						CurrentSyncGroupPicking[i] :=i;
						CurrentSyncGroupPiacing[i] :=i;
					
				
						ClipsHaveNeedle_Pick[i]:=CurrentProcessdata.PickingNeedleInfo[i].CycleStart;
					//Get placing needle info	
				END_FOR
				
				FUN_GetSyncGroup_AllocationJob(Coordinates :=CurrentPickingCoordinates,NeedleInfo:=CurrentProcessData.PickingNeedleInfo, SyncGroup=>CurrentSyncGroupPicking);
				FUN_GetSyncGroup_AllocationJob(Coordinates :=CurrentPlacingCoordinates,NeedleInfo:=CurrentProcessData.PlacingNeedleInfo, SyncGroup=>CurrentSyncGroupPiacing);
				// arrange sync group in this picking/placing job
				ClipsHaveNeedle:=ClipsHaveNeedle_Pick;
				tAutoAllocationJobBatchTimeOut.IN:=FALSE;
				AllocationJobBatchMode:=E_AllocationJob.Initial;
	
			E_AllocationJob.Initial:						
				//Get All cylinders & clips back
				bCheckTrue:=TRUE;				
				tAutoAllocationJobBatchTimeOut.IN:=TRUE	;
				
				FOR i:=0 TO NrOfAllocateCylinder - 1 DO
					clips[i].M_Retract();
					IF  clips[i].InRearPosition THEN
						cylinders[i].M_Retract();		
					END_IF	
		
					IF NOT cylinders[i].InRearPosition THEN
						bCheckTrue:=FALSE;			
					END_IF
		
				END_FOR
				// recovery Axes if error occur
				bCheckTrue:=M_RecoveryAxes();
			
				IF bCheckTrue THEN	 // Only go next step if everything is fine 
					tAutoAllocationJobBatchTimeOut.IN:=FALSE	;	
					IF bAutoAllocateJobDryRun OR SimpleAllocateMode THEN //Simple allocate mode will not placing to turn table therefor no need to check boxes on turntable						
						AllocationJobBatchMode:=E_AllocationJob.CheckRotateBeltStation;
					ELSE						
						AllocationJobBatchMode:=E_AllocationJob.CheckBoxesOnTurnTableReady;
					END_IF
					
				END_IF
				IF tAutoAllocationJobBatchTimeOut.Q THEN //Timeout error
					StatusDescription :='initiial Cylindes timeout';
					uiResumableStep := E_AllocationJob.Initial;
					_Abort :=TRUE;					
				END_IF
	
	E_AllocationJob.CheckBoxesOnTurnTableReady:
		tAutoAllocationJobBatchTimeOut.IN:=TRUE	;
		bBoxCheck:=TRUE;		
				FOR i:=0 TO 3 DO
					// if R1 or R2 used in this cycle
					IF CurrentProcessdata.PlacingNeedleInfo[i].CycleStart  THEN
						IF CurrentProcessdata.PlacingNeedleInfo[i].Box=0 THEN
							R1Used :=TRUE;
							END_IF
						
						 IF  CurrentProcessdata.PlacingNeedleInfo[i].Box=1 THEN
 							R2Used :=TRUE;
						END_IF
					END_IF

				END_FOR
				
				IF  R1Used THEN 
					  bBoxCheck :=INPUT.bTurnTable_I1Detect_Sensor AND bBoxCheck; 
				END_IF
				IF  R2Used THEN 
					  bBoxCheck := INPUT.bTurnTable_I2Detect_Sensor AND bBoxCheck; 
				END_IF
 				
				IF bBoxCheck THEN
					R1Used:=FALSE;
					R2Used:=FALSE;
					bBoxCheck :=FALSE;
					IF NOT TurnTable_Press.InFrontPosition THEN
						TurnTable_Press.M_Extend();
					END_IF
					AllocationJobBatchMode:=E_AllocationJob.CheckRotateBeltStation;
				END_IF
				
				IF tAutoAllocationJobBatchTimeOut.Q THEN
					uiResumableStep := E_AllocationJob.CheckBoxesOnTurnTableReady;
					_Abort :=TRUE	;
					StatusDescription :='Box not ready on Turn table';
				END_IF
				
	E_AllocationJob.CheckRotateBeltStation:	
		// 
		tAutoAllocationJobBatchTimeOut.IN:=FALSE;
		tAutoAllocationJobBatchTimeOut.PT := T#300S;
		
		IF ClipsHaveNeedle_Pick[iWorkingIndex] THEN
				RoundBeltMoveJob.Position:=CurrentProcessData.PickingNeedleInfo[iWorkingIndex].Station;		
				// Give RoundBelt station information
				
				IF CurrentProcessData.FastMode THEN // Fast mode : XY robot will start move to picking during rotate belt moving to request station
					IF cylinders[iWorkingCylinder].InRearPosition THEN
						arAxisCtrl_gb[AxisNo.Allocate_X].PosMode.Acc := CurrentData.Axes.Allocate_X.HalfAuto.Acceleration;
						arAxisCtrl_gb[AxisNo.Allocate_X].PosMode.Dec := CurrentData.Axes.Allocate_X.HalfAuto.Deceleration;
						arAxisCtrl_gb[AxisNo.Allocate_X].PosMode.Jerk := CurrentData.Axes.Allocate_X.HalfAuto.Jerk;
						arAxisCtrl_gb[AxisNo.Allocate_X].PosMode.Velocity := CurrentData.Axes.Allocate_X.HalfAuto.Velocity;
						arAxisCtrl_gb[AxisNo.Allocate_X].PosMode.Position := CurrentPickingCoordinates[iWorkingIndex].X;
					
						arAxisCtrl_gb[AxisNo.Allocate_Y].PosMode.Acc := CurrentData.Axes.Allocate_Y.HalfAuto.Acceleration;
						arAxisCtrl_gb[AxisNo.Allocate_Y].PosMode.Dec := CurrentData.Axes.Allocate_Y.HalfAuto.Deceleration;
						arAxisCtrl_gb[AxisNo.Allocate_Y].PosMode.Jerk := CurrentData.Axes.Allocate_Y.HalfAuto.Jerk;
						arAxisCtrl_gb[AxisNo.Allocate_Y].PosMode.Velocity := CurrentData.Axes.Allocate_Y.HalfAuto.Velocity;
						arAxisCtrl_gb[AxisNo.Allocate_Y].PosMode.Position := CurrentPickingCoordinates[iWorkingIndex].Y;						
					END_IF								
				END_IF		
				AllocationJobBatchMode:=E_AllocationJob.MovingRotateBeltStation;

			ELSE				
				AllocationJobBatchMode:=E_AllocationJob.IfNextPTP_Picking;
			END_IF

            E_AllocationJob.MovingRotateBeltStation:

              RoundBeltMoveJob.HandShake.Execute := TRUE; //Internally call rotate belt to move to request station

                IF RoundBeltMoveJob.HandShake.Busy OR RoundBeltMoveJob.HandShake.Done OR bAutoAllocateJobDryRun THEN
                  AllocationJobBatchMode := E_AllocationJob.MovedRotateBeltStation;
              END_IF
			
				IF  RoundBeltMoveJob.HandShake.Error THEN
					_Error:=TRUE;
					StatusDescription := 'Allocation batch job , Rotate belt error';
				END_IF
				AllocationJobBatchMode := E_AllocationJob.MovedRotateBeltStation;
				
            E_AllocationJob.MovedRotateBeltStation:
				// wait roundbelt object
                tAutoAllocationJobBatchTimeOut.IN := TRUE;

                bMoveRotateBeltDone := RoundBeltMoveJob.HandShake.Done;
                Ton_RoundBeltArrivedDelay.IN := bMoveRotateBeltDone;

                IF bMoveRotateBeltDone OR bAutoAllocateJobDryRun THEN
                    RoundBeltMoveJob.HandShake.Execute := FALSE;
                    tAutoAllocationJobBatchTimeOut.IN := FALSE;
                    AllocationJobBatchMode := E_AllocationJob.MoveToTargetPos;
                END_IF

                IF tAutoAllocationJobBatchTimeOut.Q THEN
                    StatusDescription := 'Rotate Belt TimeOut';
                    uiResumableStep := E_AllocationJob.MovingRotateBeltStation;
                    _Abort           := TRUE;
                END_IF
				
					
            E_AllocationJob.MoveToTargetPos:
                Ton_RoundBeltArrivedDelay.IN := FALSE;
                tAutoAllocationJobBatchTimeOut.IN := TRUE;

                iWorkingCylinder :=CurrentProcessData.PickingNeedleInfo[iWorkingIndex].Clip ;

                IF NOT CurrentProcessData.FastMode THEN
					IF cylinders[iWorkingCylinder].InRearPosition THEN							
						arAxisCtrl_gb[AxisNo.Allocate_X].PosMode.Acc := CurrentData.Axes.Allocate_X.HalfAuto.Acceleration;
						arAxisCtrl_gb[AxisNo.Allocate_X].PosMode.Dec := CurrentData.Axes.Allocate_X.HalfAuto.Deceleration;
						arAxisCtrl_gb[AxisNo.Allocate_X].PosMode.Jerk := CurrentData.Axes.Allocate_X.HalfAuto.Jerk;
						arAxisCtrl_gb[AxisNo.Allocate_X].PosMode.Velocity := CurrentData.Axes.Allocate_X.HalfAuto.Velocity;
						arAxisCtrl_gb[AxisNo.Allocate_X].PosMode.Position := CurrentPickingCoordinates[iWorkingIndex].X;
					
						arAxisCtrl_gb[AxisNo.Allocate_Y].PosMode.Acc := CurrentData.Axes.Allocate_Y.HalfAuto.Acceleration;
						arAxisCtrl_gb[AxisNo.Allocate_Y].PosMode.Dec := CurrentData.Axes.Allocate_Y.HalfAuto.Deceleration;
						arAxisCtrl_gb[AxisNo.Allocate_Y].PosMode.Jerk := CurrentData.Axes.Allocate_Y.HalfAuto.Jerk;
						arAxisCtrl_gb[AxisNo.Allocate_Y].PosMode.Velocity := CurrentData.Axes.Allocate_Y.HalfAuto.Velocity;
						arAxisCtrl_gb[AxisNo.Allocate_Y].PosMode.Position := CurrentPickingCoordinates[iWorkingIndex].Y;	
					END_IF
                END_IF

                IF (arAxisCtrl_gb[AxisNo.Allocate_X].Admin.Axis.Status.Moving OR  
			(arAxisStatus_gb[AxisNo.Allocate_X].Admin._OpModeAck = ModePosAbs AND arAxisStatus_gb[AxisNo.Allocate_X].Admin.CmdDone) )AND  
					(arAxisCtrl_gb[AxisNo.Allocate_Y].Admin.Axis.Status.Moving OR 
					(arAxisStatus_gb[AxisNo.Allocate_Y].Admin._OpModeAck = ModePosAbs AND arAxisStatus_gb[AxisNo.Allocate_Y].Admin.CmdDone))
					(* AND RoundBelt.AllocatingArea.PressCylinder.InFrontPosition *) THEN
					tAutoAllocationJobBatchTimeOut.IN := FALSE;
                    AllocationJobBatchMode := E_AllocationJob.MovingToTargetPos;
                END_IF
 				
				IF arAxisCtrl_gb[AxisNo.Allocate_Y].Admin.Axis.Status.Error AND 
					arAxisCtrl_gb[AxisNo.Allocate_X].Admin.Axis.Status.Error  THEN
					_Error :=TRUE;
					StatusDescription :='Allocate robot error';
				END_IF
				
				 IF tAutoAllocationJobBatchTimeOut.Q THEN

                    StatusDescription := 'Allocate robot TimeOut';
                    uiResumableStep := E_AllocationJob.MoveToTargetPos;
                    _Abort           := TRUE;

                END_IF
				
            E_AllocationJob.MovingToTargetPos:

                tAutoAllocationJobBatchTimeOut.IN := TRUE;

                IF (arAxisStatus_gb[AxisNo.Allocate_Y].Admin._OpModeAck = ModePosAbs AND arAxisStatus_gb[AxisNo.Allocate_Y].Admin.CmdDone) AND 
					(arAxisStatus_gb[AxisNo.Allocate_X].Admin._OpModeAck = ModePosAbs AND arAxisStatus_gb[AxisNo.Allocate_X].Admin.CmdDone) THEN
                    tAutoAllocationJobBatchTimeOut.IN := FALSE;
					IF bAutoAllocateJobDryRun THEN
                   	 AllocationJobBatchMode                := E_AllocationJob.CylinderDownPick;
					ELSE
						AllocationJobBatchMode             := E_AllocationJob.CheckBoxReadyOnAllocatePosOfRoundBelt;
					END_IF
                END_IF

                IF tAutoAllocationJobBatchTimeOut.Q THEN
                    StatusDescription := 'Moving to picking position timeout';
                    uiResumableStep := E_AllocationJob.MoveToTargetPos;
                    _Abort           := TRUE;
                END_IF
				
				
			E_AllocationJob.CheckBoxReadyOnAllocatePosOfRoundBelt:
				tAutoAllocationJobBatchTimeOut.IN:=TRUE	;
				bBoxCheck :=TRUE;
				FOR i:=0 TO 3 DO //Check if request box is on the belt 
					IF CurrentProcessData.PickingNeedleInfo[i].Station =  CurrentProcessData.PickingNeedleInfo[iWorkingIndex].Station THEN
						IF CurrentProcessData.PickingNeedleInfo[i].Box=0   THEN
							A1Used :=TRUE;
							END_IF
						
						 IF  CurrentProcessData.PickingNeedleInfo[i].Box=1 THEN
 							A2Used :=TRUE;
						END_IF
					END_IF
				END_FOR
				
				IF  A1Used THEN 
					  bBoxCheck :=INPUT.bRoundBelt_WorkZoneQ1Detect_Sensor AND bBoxCheck; 
				END_IF
				IF  A2Used THEN 
					  bBoxCheck :=INPUT.bRoundBelt_WorkZoneQ2Detect_Sensor AND bBoxCheck; 
				END_IF
 				
				IF bBoxCheck THEN
						bBoxCheck:=A1Used:=A2Used:=FALSE;
						tAutoAllocationJobBatchTimeOut.IN:=FALSE	;
						IF RoundBelt_Press.InFrontPosition THEN
							AllocationJobBatchMode:=E_AllocationJob.CylinderDownPick;
						ELSE
							//RoundBelt_Press.M_Extend();	
						END_IF
				END_IF
				
				IF tAutoAllocationJobBatchTimeOut.Q THEN
					_Abort :=TRUE	;
					uiResumableStep :=E_AllocationJob.CheckBoxReadyOnAllocatePosOfRoundBelt;
					StatusDescription :='Box not ready on Rotate Belt';
				END_IF

            E_AllocationJob.CylinderDownPick:
                
                bCylinderCheck:=TRUE;
				tAutoAllocationJobBatchTimeOut.IN := TRUE;       
				
				
                THIS^.cylinders[iWorkingCylinder].M_Extend();//'AutoMode E_AllocationJob.CylinderDownPick');
				// Cylinder move down
				
				IF CurrentProcessData.SyncMode THEN
					///Sync mode : all clips in same sync group will move together to picking / placing
					FOR i := iWorkingIndex+1 TO 3 DO
						IF CurrentSyncGroupPicking[i]=CurrentSyncGroupPicking[iWorkingIndex] AND 
							ClipsHaveNeedle_Pick[i]	 THEN
							cylinders[CurrentProcessData.PickingNeedleInfo[i].Clip].M_Extend();//'Auto Mode E_AllocationJob.CylinderDownPick in Sync picking Mode');
							bCylinderCheck :=cylinders[CurrentProcessData.PickingNeedleInfo[i].Clip].InFrontPosition AND bCylinderCheck;			
						END_IF
					END_FOR
					
				END_IF
                
                IF cylinders[iWorkingCylinder].InFrontPosition AND bCylinderCheck THEN
                    tAutoAllocationJobBatchTimeOut.IN := FALSE;
                    AllocationJobBatchMode                := E_AllocationJob.ClipColse;
                END_IF

                IF tAutoAllocationJobBatchTimeOut.Q THEN

                    StatusDescription := 'Picking down timeout';
                    _Abort :=TRUE	;
					uiResumableStep :=E_AllocationJob.CylinderDownPick;

                END_IF

            E_AllocationJob.ClipColse:
                Ton_RoundBeltArrivedDelay.IN := FALSE;
                tAutoAllocationJobBatchTimeOut.IN := TRUE;
				bCylinderCheck:=TRUE;
				
                THIS^.clips[iWorkingCylinder].M_Extend();//'Auto Mode E_AllocationJob.ClipColse');
				IF CurrentProcessData.SyncMode THEN
					FOR i := iWorkingIndex+1 TO 3 DO
						IF CurrentSyncGroupPicking[i]=CurrentSyncGroupPicking[iWorkingIndex] AND 
							ClipsHaveNeedle_Pick[i]	 THEN
							clips[CurrentProcessData.PickingNeedleInfo[i].Clip].M_Extend();//'Auto Mode E_AllocationJob.ClipColse in Sync pick Mode');
							bCylinderCheck :=clips[CurrentProcessData.PickingNeedleInfo[i].Clip].InFrontPosition AND bCylinderCheck;			
						END_IF
					END_FOR
					
				END_IF
				
                IF clips[iWorkingCylinder].InFrontPosition AND bCylinderCheck THEN
                    tAutoAllocationJobBatchTimeOut.IN := FALSE;
                    AllocationJobBatchMode                := E_AllocationJob.CylinderUpPick;
                END_IF

                IF tAutoAllocationJobBatchTimeOut.Q THEN

                    StatusDescription := 'Picking Close timeout';
                    _Error := TRUE;

                END_IF

	E_AllocationJob.CylinderUpPick:
		bCylinderCheck:=TRUE;
		//bCylinderCheckFastMode:=TRUE;					
		bBoxCheck :=TRUE;
		
		tAutoAllocationJobBatchTimeOut.IN:=TRUE	;
		
		THIS^.cylinders[iWorkingCylinder].M_Retract();// 'Auto Mode E_AllocationJob.CylinderUpPick');		
		
		IF CurrentProcessData.SyncMode THEN
					FOR i := iWorkingIndex+1 TO 3 DO
						IF CurrentSyncGroupPicking[i]=CurrentSyncGroupPicking[iWorkingIndex] AND 
							ClipsHaveNeedle_Pick[i]	 THEN
							cylinders[CurrentProcessData.PickingNeedleInfo[i].Clip].M_Retract();// 'Auto Mode E_AllocationJob.CylinderUpPick in Sync pick Mode');
							bCylinderCheck :=cylinders[CurrentProcessData.PickingNeedleInfo[i].Clip].InRearPosition AND bCylinderCheck;
							//bCylinderCheckFastMode := (NOT cylinders[CurrentProcessData.PickingNeedleInfo[i].Clip].InFrontPosition) AND bCylinderCheckFastMode;
						END_IF
					END_FOR
					
		END_IF
		
				IF  A1Used THEN 
					  bBoxCheck :=INPUT.bRoundBelt_WorkZoneQ1Detect_Sensor AND bBoxCheck; 
				END_IF
				IF  A2Used THEN 
					  bBoxCheck :=INPUT.bRoundBelt_WorkZoneQ2Detect_Sensor AND bBoxCheck; 
				END_IF
				//Check if box still there
				
(*//====	2026/03/31 取消fastmode		edited by Gamin
		IF CurrentProcessData.FastMode AND bCylinderCheckFastMode AND (NOT cylinders[iWorkingCylinder].InFrontPosition) THEN
			tonFastModeTimeDelayBatch.IN:=TRUE;
		END_IF
		
		IF (cylinders[iWorkingCylinder].InRearPosition AND bCylinderCheck )OR  tonFastModeTimeDelayBatch.Q  THEN
			//Fast mode : go next step when cylinder is leave the front sensor with certain time delay
				tonFastModeTimeDelayBatch.IN:=FALSE;			
				AllocationJobBatchMode:=E_AllocationJob.IfNextPTP_Picking;
		END_IF
==========================*)
				IF cylinders[iWorkingCylinder].InRearPosition AND bCylinderCheck THEN
					AllocationJobBatchMode:=E_AllocationJob.IfNextPTP_Picking;
				END_IF

		IF tAutoAllocationJobBatchTimeOut.Q THEN			
			StatusDescription :='Picking Up timeout';
			_Abort :=TRUE	;
			uiResumableStep :=E_AllocationJob.CylinderUpPick;
		END_IF
		
	E_AllocationJob.IfNextPTP_Picking:
		tAutoAllocationJobBatchTimeOut.IN:=FALSE	;	
		iPickingNeedleCount:=1;
			FOR i := iWorkingIndex+1 TO 3 DO //remove request if already processed in previous sync group
				IF CurrentSyncGroupPicking[i]=CurrentSyncGroupPicking[iWorkingIndex] AND 
				   ClipsHaveNeedle_Pick[i]	 THEN
						iPickingNeedleCount:=iPickingNeedleCount+1;
						ClipsHaveNeedle_Pick[i]:=FALSE;		
				END_IF
			END_FOR
			
		iWorkingIndex:=iWorkingIndex+1;
		IF iWorkingIndex>= NrOfAllocateCylinder THEN //All picking job done in this cycle , go to placing processing
			iWorkingIndex:=0;
			tAutoAllocationJobBatchTimeOut.IN:=FALSE	;
			IF SimpleAllocateMode THEN //If Simple allocate mode , need to check the target box is ready on rotate belt
				AllocationJobBatchMode:=E_AllocationJob.CheckRotateBeltStation_SimpleAllocatePlacing;
			ELSE
				AllocationJobBatchMode:=E_AllocationJob.MoveToPlacingPos;
			END_IF
		ELSE
			
			AllocationJobBatchMode:=E_AllocationJob.CheckRotateBeltStation;		
			 //Still picking job
		END_IF
		
	

	E_AllocationJob.CheckRotateBeltStation_SimpleAllocatePlacing:	
		// Check if the Rotate belt is in the target.
		tAutoAllocationJobBatchTimeOut.IN:=FALSE;		
		IF ClipsHaveNeedle[iWorkingIndex] THEN
			RoundBeltMoveJob.Position:=CurrentProcessData.PlacingNeedleInfo[iWorkingIndex].Station;	
			// Give roundBelt station
			AllocationJobBatchMode:=E_AllocationJob.MovingRotateBeltStation_SimpleAllocatePlacing;
				IF CurrentProcessData.FastMode THEN // Fast mode : XY robot will start move to picking during rotate belt moving to request station
					IF cylinders[iWorkingCylinder].InRearPosition THEN				
						arAxisCtrl_gb[AxisNo.Allocate_X].PosMode.Acc := CurrentData.Axes.Allocate_X.HalfAuto.Acceleration;
						arAxisCtrl_gb[AxisNo.Allocate_X].PosMode.Dec := CurrentData.Axes.Allocate_X.HalfAuto.Deceleration;
						arAxisCtrl_gb[AxisNo.Allocate_X].PosMode.Jerk := CurrentData.Axes.Allocate_X.HalfAuto.Jerk;
						arAxisCtrl_gb[AxisNo.Allocate_X].PosMode.Velocity := CurrentData.Axes.Allocate_X.HalfAuto.Velocity;
						arAxisCtrl_gb[AxisNo.Allocate_X].PosMode.Position := CurrentPlacingCoordinates[iWorkingIndex].X;
					
						arAxisCtrl_gb[AxisNo.Allocate_Y].PosMode.Acc := CurrentData.Axes.Allocate_Y.HalfAuto.Acceleration;
						arAxisCtrl_gb[AxisNo.Allocate_Y].PosMode.Dec := CurrentData.Axes.Allocate_Y.HalfAuto.Deceleration;
						arAxisCtrl_gb[AxisNo.Allocate_Y].PosMode.Jerk := CurrentData.Axes.Allocate_Y.HalfAuto.Jerk;
						arAxisCtrl_gb[AxisNo.Allocate_Y].PosMode.Velocity := CurrentData.Axes.Allocate_Y.HalfAuto.Velocity;
						arAxisCtrl_gb[AxisNo.Allocate_Y].PosMode.Position := CurrentPlacingCoordinates[iWorkingIndex].Y;						
					END_IF							
				END_IF
		
			ELSE
				
				AllocationJobBatchMode:=E_AllocationJob.IfNextPTP_Placing;
			END_IF

            E_AllocationJob.MovingRotateBeltStation_SimpleAllocatePlacing:

                

                RoundBeltMoveJob.HandShake.Execute := TRUE; //Internally call rotate belt to move to request station

                IF RoundBeltMoveJob.HandShake.Busy OR RoundBeltMoveJob.HandShake.Done OR bAutoAllocateJobDryRun THEN
                    AllocationJobBatchMode := E_AllocationJob.MovedRotateBeltStation_SimpleAllocatePlacing;
                END_IF
				
				IF  RoundBeltMoveJob.HandShake.Error THEN
					_Error:=TRUE;
					StatusDescription := 'Allocation batch job , Rotate belt error';
				END_IF

            E_AllocationJob.MovedRotateBeltStation_SimpleAllocatePlacing:

                tAutoAllocationJobBatchTimeOut.IN := TRUE;

                bMoveRotateBeltDone := RoundBeltMoveJob.HandShake.Done;
                Ton_RoundBeltArrivedDelay.IN := bMoveRotateBeltDone;

                IF bMoveRotateBeltDone OR bAutoAllocateJobDryRun THEN
                    RoundBeltMoveJob.HandShake.Execute := FALSE;
                	tAutoAllocationJobBatchTimeOut.IN := FALSE;
                    AllocationJobBatchMode := E_AllocationJob.CheckBoxReadyOnRoundBelt_SimpleAllocateMode;
                END_IF

                IF tAutoAllocationJobBatchTimeOut.Q THEN
                    StatusDescription := 'Rotate Belt TimeOut';
                    uiResumableStep := E_AllocationJob.MovingRotateBeltStation_SimpleAllocatePlacing;
                    _Abort           := TRUE;
                END_IF
				
	E_AllocationJob.CheckBoxReadyOnRoundBelt_SimpleAllocateMode:
		tAutoAllocationJobBatchTimeOut.IN:=TRUE	;
				bBoxCheck :=TRUE;
				FOR i:=0 TO 3 DO //Check if request box is on the belt 					
						IF CurrentProcessData.PlacingNeedleInfo[i].Box=0   THEN
							A1Used :=TRUE;
							END_IF
						
						 IF  CurrentProcessData.PlacingNeedleInfo[i].Box=1 THEN
 							A2Used :=TRUE;
						END_IF
					
				END_FOR
				
				IF  A1Used THEN 
					  bBoxCheck :=INPUT.bRoundBelt_WorkZoneQ1Detect_Sensor AND bBoxCheck; 
				END_IF
				IF  A2Used THEN 
					  bBoxCheck :=INPUT.bRoundBelt_WorkZoneQ2Detect_Sensor AND bBoxCheck; 
				END_IF
 				
				IF bBoxCheck THEN
						bBoxCheck:=A1Used:=A2Used:=FALSE;
						tAutoAllocationJobBatchTimeOut.IN:=FALSE;
						AllocationJobBatchMode:=E_AllocationJob.MoveToPlacingPos;
				END_IF
				
				IF tAutoAllocationJobBatchTimeOut.Q THEN
					_Abort :=TRUE	;
					uiResumableStep :=E_AllocationJob.CheckBoxReadyOnRoundBelt_SimpleAllocateMode;
					StatusDescription :='Box not ready on Rotate Belt ';
				END_IF			
	
     E_AllocationJob.MoveToPlacingPos:
                
				tAutoAllocationJobBatchTimeOut.IN:=TRUE;
                IF ClipsHaveNeedle[iWorkingIndex] THEN 
                    iWorkingCylinder := CurrentProcessData.PlacingNeedleInfo[iWorkingIndex].Clip;
					IF cylinders[iWorkingCylinder].InRearPosition THEN
						arAxisCtrl_gb[AxisNo.Allocate_X].PosMode.Acc := CurrentData.Axes.Allocate_X.HalfAuto.Acceleration;
						arAxisCtrl_gb[AxisNo.Allocate_X].PosMode.Dec := CurrentData.Axes.Allocate_X.HalfAuto.Deceleration;
						arAxisCtrl_gb[AxisNo.Allocate_X].PosMode.Jerk := CurrentData.Axes.Allocate_X.HalfAuto.Jerk;
						arAxisCtrl_gb[AxisNo.Allocate_X].PosMode.Velocity := CurrentData.Axes.Allocate_X.HalfAuto.Velocity;
						arAxisCtrl_gb[AxisNo.Allocate_X].PosMode.Position := CurrentPlacingCoordinates[iWorkingIndex].X;
					
						arAxisCtrl_gb[AxisNo.Allocate_Y].PosMode.Acc := CurrentData.Axes.Allocate_Y.HalfAuto.Acceleration;
						arAxisCtrl_gb[AxisNo.Allocate_Y].PosMode.Dec := CurrentData.Axes.Allocate_Y.HalfAuto.Deceleration;
						arAxisCtrl_gb[AxisNo.Allocate_Y].PosMode.Jerk := CurrentData.Axes.Allocate_Y.HalfAuto.Jerk;
						arAxisCtrl_gb[AxisNo.Allocate_Y].PosMode.Velocity := CurrentData.Axes.Allocate_Y.HalfAuto.Velocity;
						arAxisCtrl_gb[AxisNo.Allocate_Y].PosMode.Position := CurrentPlacingCoordinates[iWorkingIndex].Y;						
					END_IF
							
					IF CurrentProcessData.FastMode AND NOT SimpleAllocateMode THEN // Fast mode : When robot go to placing needles , Rotatebelt will start to move to next picking station	But not allow in simple allocate job due to placing location is rotatebelt also					
						IF AutoAllocateJobBatch_Ctrl.AutoMode_AllocateMoveBatch.NrOfAllocationJob > iProcessingIndex+1 THEN//AND AutoAllocateJobBatch_Ctrl.AutoMode_AllocateMoveBatch.AllocationInfo[iProcessingIndex+1]. <> iCurrentRotateBeltStation THEN
							FOR i := 0 TO 3 DO 
								IF	AutoAllocateJobBatch_Ctrl.AutoMode_AllocateMoveBatch.AllocationInfo[iProcessingIndex+1].PickingNeedleInfo[i].CycleStart THEN
									iNextPickingStation :=   AutoAllocateJobBatch_Ctrl.AutoMode_AllocateMoveBatch.AllocationInfo[iProcessingIndex+1].PickingNeedleInfo[i].Station;
									bIfNextCycle:=TRUE;
									EXIT;
								END_IF
							END_FOR
						END_IF					
					END_IF							
							

                    IF (arAxisCtrl_gb[AxisNo.Allocate_X].Admin.Axis.Status.Moving AND  arAxisCtrl_gb[AxisNo.Allocate_Y].Admin.Axis.Status.Moving) OR
 						(arAxisStatus_gb[AxisNo.Allocate_X].Admin._OpModeAck = ModePosAbs AND arAxisStatus_gb[AxisNo.Allocate_X].Admin.CmdDone) AND 
						(arAxisStatus_gb[AxisNo.Allocate_Y].Admin._OpModeAck = ModePosAbs AND arAxisStatus_gb[AxisNo.Allocate_Y].Admin.CmdDone) THEN
						bIfNextCycle :=FALSE;
						tAutoAllocationJobBatchTimeOut.IN:=FALSE	;
                        AllocationJobBatchMode := E_AllocationJob.MovingToPlacingPos;
                    END_IF

                ELSE

                    AllocationJobBatchMode := E_AllocationJob.IfNextPTP_Placing;
                END_IF
				
				IF tAutoAllocationJobBatchTimeOut.Q THEN
			
					StatusDescription :='Move to placing timeout';
					uiResumableStep := E_AllocationJob.MoveToPlacingPos;
					_Abort := TRUE;
					
				END_IF

            E_AllocationJob.MovingToPlacingPos:

                tAutoAllocationJobBatchTimeOut.IN := TRUE;

					IF (arAxisStatus_gb[AxisNo.Allocate_X].Admin._OpModeAck = ModePosAbs AND arAxisStatus_gb[AxisNo.Allocate_X].Admin.CmdDone) AND 
						(arAxisStatus_gb[AxisNo.Allocate_Y].Admin._OpModeAck = ModePosAbs AND arAxisStatus_gb[AxisNo.Allocate_Y].Admin.CmdDone) THEN
                    tAutoAllocationJobBatchTimeOut.PT := T#300S;
                    tAutoAllocationJobBatchTimeOut.IN := FALSE;
                    AllocationJobBatchMode                := E_AllocationJob.CylinderDownPlace;
                END_IF

                IF tAutoAllocationJobBatchTimeOut.Q THEN
                    StatusDescription := 'Moving placing timeout';
                    uiResumableStep := E_AllocationJob.MoveToPlacingPos;
                    _Abort           := TRUE;

                END_IF

            E_AllocationJob.CylinderDownPlace:
				bCylinderCheck:=TRUE;
                tAutoAllocationJobBatchTimeOut.IN := TRUE;
                cylinders[iWorkingCylinder].M_Extend();//'Auto Mode E_AllocationJob.CylinderDownPlace');
				
				IF CurrentProcessData.SyncMode THEN
					FOR i := iWorkingIndex+1 TO 3 DO
						IF CurrentSyncGroupPiacing[i]=CurrentSyncGroupPiacing[iWorkingIndex] AND 
							ClipsHaveNeedle[i]	 THEN
							cylinders[CurrentProcessData.PlacingNeedleInfo[i].Clip].M_Extend();//'Auto Mode E_AllocationJob.CylinderDownPlace in Sync placing Mode');
							bCylinderCheck :=cylinders[CurrentProcessData.PlacingNeedleInfo[i].Clip ].InFrontPosition AND bCylinderCheck;			
						END_IF
					END_FOR
					
				END_IF
				
               	 IF cylinders[iWorkingCylinder].InFrontPosition AND bCylinderCheck THEN
                    tAutoAllocationJobBatchTimeOut.IN := FALSE;
                    AllocationJobBatchMode            := E_AllocationJob.ClipOpen;
              	  END_IF
				
                IF tAutoAllocationJobBatchTimeOut.Q THEN

                    StatusDescription := ' placing down timeout';
                   _Abort :=TRUE	;
					uiResumableStep :=E_AllocationJob.CylinderDownPlace;

                END_IF

            E_AllocationJob.ClipOpen:
                tAutoAllocationJobBatchTimeOut.IN := TRUE;
				bCylinderCheck:=TRUE;
                clips[iWorkingCylinder].M_Retract();// 'Auto Mode E_AllocationJob.ClipOpen');
					IF CurrentProcessData.SyncMode THEN
					FOR i := iWorkingIndex+1 TO 3 DO
						IF CurrentSyncGroupPiacing[i]=CurrentSyncGroupPiacing[iWorkingIndex] AND 
							ClipsHaveNeedle[i]	 THEN
							clips[CurrentProcessData.PlacingNeedleInfo[i].Clip].M_Retract();// 'Auto Mode E_AllocationJob.ClipOpen in Sync placing Mode');
							bCylinderCheck :=clips[CurrentProcessData.PlacingNeedleInfo[i].Clip].InRearPosition AND bCylinderCheck;			
						END_IF
					END_FOR
					
				END_IF
				
				
                IF clips[iWorkingCylinder].InRearPosition AND bCylinderCheck THEN
                    tAutoAllocationJobBatchTimeOut.IN := FALSE;
                    AllocationJobBatchMode                := E_AllocationJob.CylinderUpPlace;
                END_IF

                IF tAutoAllocationJobBatchTimeOut.Q THEN

                    StatusDescription := ' placing Open timeout';
                    _Error := TRUE;

                END_IF

            E_AllocationJob.CylinderUpPlace:
				bCylinderCheck:=TRUE;
				//bCylinderCheckFastMode:=TRUE;
				tAutoAllocationJobBatchTimeOut.IN:=TRUE;
				
                cylinders[iWorkingCylinder].M_Retract();// ' Auto Mode E_AllocationJob.CylinderUpPlace');
				
					IF CurrentProcessData.SyncMode THEN
					FOR i := iWorkingIndex+1 TO 3 DO
						IF CurrentSyncGroupPiacing[i]=CurrentSyncGroupPiacing[iWorkingIndex] AND 
							ClipsHaveNeedle[i]	 THEN
							cylinders[CurrentProcessData.PlacingNeedleInfo[i].Clip].M_Retract();// 'Auto Mode E_AllocationJob.CylinderUpPlace in Sync placing Mode');
							bCylinderCheck :=cylinders[CurrentProcessData.PlacingNeedleInfo[i].Clip ].InRearPosition AND bCylinderCheck;	
							//bCylinderCheckFastMode := (NOT cylinders[CurrentProcessData.PlacingNeedleInfo[i].Clip ].InFrontPosition) AND bCylinderCheckFastMode ;
							
						END_IF
					END_FOR					
				END_IF
(*================	取消 fastmode，防止偷跑導致撞機，edited BY Gamin 2026/03/31
				IF CurrentProcessData.FastMode  AND (NOT cylinders[iWorkingCylinder].InFrontPosition) AND bCylinderCheckFastMode THEN						
               		 tonFastModeTimeDelayBatch.IN := TRUE;
				END_IF
				
                IF (cylinders[iWorkingCylinder].InRearPosition AND bCylinderCheck) OR tonFastModeTimeDelayBatch.Q THEN
                    tAutoAllocationJobBatchTimeOut.IN         := FALSE;
					tonFastModeTimeDelayBatch.IN 				  := FALSE;
                    
                    AllocationJobBatchMode := E_AllocationJob.CheckNeedlePlaced;
                END_IF
====================*)
				IF cylinders[iWorkingCylinder].InRearPosition AND bCylinderCheck THEN
                    tAutoAllocationJobBatchTimeOut.IN         := FALSE;
                    AllocationJobBatchMode := E_AllocationJob.CheckNeedlePlaced;
                END_IF
				
                IF tAutoAllocationJobBatchTimeOut.Q THEN

                    StatusDescription := ' placing Up timeout';
                    _Abort :=TRUE	;
					uiResumableStep :=E_AllocationJob.CylinderUpPlace;

                END_IF

			E_AllocationJob.CheckNeedlePlaced:
				ClipsHaveNeedle[iWorkingIndex] :=FALSE;
					IF CurrentProcessData.SyncMode THEN
					FOR i := iWorkingIndex+1 TO 3 DO
						IF CurrentSyncGroupPiacing[i]=CurrentSyncGroupPiacing[iWorkingIndex] AND 
							ClipsHaveNeedle[i]	 THEN
							ClipsHaveNeedle[i]:=FALSE;
							
						END_IF
					END_FOR		
				END_IF
				
				
				AllocationJobBatchMode := E_AllocationJob.IfNextPTP_Placing;
				
            E_AllocationJob.IfNextPTP_Placing:
                iWorkingIndex := iWorkingIndex + 1;

                IF iWorkingIndex >= NrOfAllocateCylinder THEN
                    iWorkingIndex := 0;
                    AllocationJobBatchMode := E_AllocationJob.Finish;
                ELSE
					IF SimpleAllocateMode THEN
						AllocationJobBatchMode := E_AllocationJob.CheckRotateBeltStation_SimpleAllocatePlacing;
					ELSE
                    	AllocationJobBatchMode := E_AllocationJob.MoveToPlacingPos;
               	 END_IF
				END_IF        

            E_AllocationJob.Finish:
                // Finish
					//Update needling data
					arrProcessedIndex[iProcessingIndex] :=CurrentProcessData.ID;
				IF 	AutoAllocateJobBatch_Ctrl.AutoMode_AllocateMoveBatch.NrOfAllocationJob> iProcessingIndex THEN

					iProcessingIndex :=iProcessingIndex+1;
					AllocationJobBatchMode := E_AllocationJob.PreDataProcess;
				ELSE
					// 最後一筆邏輯完成,但機械可能還在收尾。
					// 進入 FinalCleanup gate,等所有 cylinder/clip/press 都歸位、RoundBelt idle 才設 _Executed
					AllocationJobBatchMode := E_AllocationJob.FinalCleanup;
				END_IF

			E_AllocationJob.FinalCleanup:
				// 給 Done 之前的最終收尾 gate:
				// 確保整批做完後,所有 cylinder/clip 都退到安全位置、RoundBelt 不再 Busy,
				// 才允許 _Executed := TRUE → STATE_DONE。
				// 目的: 上位看到 Done 時、PLC 內部資料(ProcessedIndex/WorkedID)跟機械都已穩定,
				//       上位撤 Execute 後即使馬上下一包進來也不會撞到上一包未收尾的狀態。
				// 註: TurnTable_Press / RoundBelt_Press 不收 — 兩個 Press 只是壓住盒子,
				//     對下一批的 X/Y robot 跟 cylinder 升降都沒有安全顧慮;
				//     收了反而會讓盒子晃動,且下一批 CheckBoxesOnTurnTableReady 還要再 Extend。
				tAutoAllocationJobBatchTimeOut(IN := TRUE, PT := T#10S);
				bCheckTrue := TRUE;

				FOR i := 0 TO NrOfAllocateCylinder-1 DO
					clips[i].M_Retract();
					IF clips[i].InRearPosition THEN
						cylinders[i].M_Retract();
					END_IF
					IF NOT cylinders[i].InRearPosition OR NOT clips[i].InRearPosition THEN
						bCheckTrue := FALSE;
					END_IF
				END_FOR

				// 圓帶不可還在動作中
				IF RoundBeltMoveJob_Status.Busy THEN
					bCheckTrue := FALSE;
				END_IF

				// 同步把最後一筆 ID 確實出到 ProcessedIndex (頂部已每 cycle 拷貝,這裡是雙保險)
				ProcessedIndex := arrProcessedIndex;

				IF bCheckTrue THEN
					tAutoAllocationJobBatchTimeOut.IN := FALSE;
					_Executed := TRUE;
				END_IF

				IF tAutoAllocationJobBatchTimeOut.Q THEN
					StatusDescription := 'FinalCleanup timeout: hardware not back to safe position';
					_UniqueErrorCode := 'E_FINAL_CLEANUP_TIMEOUT';
					uiResumableStep := E_AllocationJob.FinalCleanup;
					_Abort := TRUE;
				END_IF

        END_CASE

IF NOT Execute THEN
	eState:=STATE_RESETTING;
END_IF
IF _Error THEN
	eState:=STATE_ERROR;
END_IF
IF _Abort THEN
	eSTATE:=STATE_ABORTING;
END_IF
IF _Executed THEN
	eSTATE:=STATE_Done;
END_IF
END_METHOD

METHOD  M_STATE_RESETTING
VAR_INPUT
END_VAR
VAR	
	bCylinderCheck : BOOL;
END_VAR
Busy                         := TRUE;
Error                        := _Error;
tAutoAllocationJobBatchTimeOut.IN := FALSE;

  CASE uiResettingStep OF
            0:
                // Resetting process start

                uiAbortingStep := 0;
                uiAbortedStep  := 0;
				_bRetry := FALSE;
				RoundBeltMoveJob.HandShake.Execute:=FALSE;
				RoundBeltMoveJob_Ctrl.Execute:= RoundBeltMoveJob.HandShake.Execute;
				DAS_CoreSys.MachineControl.fbAllocateArea.M_ReleaseRoundBeltAccess(E_RoundBeltControlAccess.Allocating);

                IF M_RecoveryAxes() THEN
					uiResettingStep := 1000;
				END_IF

            1000:
				bCylinderCheck :=TRUE;
//                FOR i := 1 TO 3 DO
//                    IF cylinders[i].xError THEN
//                         cylinders[i].M_Reset();
//						 ELSE
//						 cylinders[i].M_Retract();
//                    END_IF
//				bCylinderCheck := bCylinderCheck AND cylinders[i].InRearPosition;

//                END_FOR
				RoundBeltMoveJob.HandShake.Execute:=FALSE;
				RoundBeltMoveJob_Ctrl.Execute:= RoundBeltMoveJob.HandShake.Execute;
				DAS_CoreSys.MachineControl.fbAllocateArea.M_ReleaseRoundBeltAccess(E_RoundBeltControlAccess.Allocating);
                uiResettingStep := 2000;

			2000:
//					IF TurnTable.Motor.Error THEN
//					TurnTable.Motor.Reset();
//				END_IF

//				IF  AllocateRobot.axX.Error THEN
//					  AllocateRobot.axX.Reset();
//				END_IF

//				IF  AllocateRobot.axY.Error THEN
//					  AllocateRobot.axY.Reset();
//				END_IF

//				IF RoundBelt.Motor.Error THEN
//					RoundBelt.Motor.Reset();
//				END_IF
				uiResettingStep := 9000;

            9000:
                // Resetting process is finished
                Done := FALSE;
                Busy := FALSE;
                bResettingCompleted := TRUE;
        END_CASE

        IF bResettingCompleted THEN
            eState := STATE_DORMANT;
        END_IF
END_METHOD

END_FUNCTION_BLOCK

// ---- POUs/DAS_CoreSys.TcPOU
PROGRAM DAS_CoreSys
VAR
    UserModeCofig  : PML_UnitModeConfig; //User can configure his own Mode
    MachineControl : FB_MachineControl;
	CoreSys_Stop : BOOL;
	CoreSys_Reset :BOOL;
	CoreSys_Start : BOOL;
	CoreSys_Estop : BOOL;
	OP_Mode : E_UnitMode := E_UnitMode.Manual;
	trigResetForRS485 : R_TRIG;
END_VAR

A00_BasicUnit();
A10_StatusCtrl();


CASE GVL_ADS.MachineMode.TargetMode OF
		E_MachineMode.MANUAL:
			OP_Mode := E_UnitMode.Manual;
		E_MachineMode.AUTO:
			OP_Mode := E_UnitMode.Auto;
ELSE
	OP_Mode := E_UnitMode.Manual;
END_CASE


//IF OP_Mode = E_UnitMode.Manual THEN
//	GVL_ADS.MachineMode.CurrentMode := E_MachineMode.MANUAL;
//ELSIF OP_Mode = E_UnitMode.Auto AND MachineControl.MachineHomed THEN
	
//	GVL_ADS.MachineMode.CurrentMode := E_MachineMode.AUTO;
//END_IF

IF PackTags[0].Status.UnitModeCurrent = E_UnitMode.Manual THEN
	GVL_ADS.MachineMode.CurrentMode := E_MachineMode.MANUAL;
ELSIF PackTags[0].Status.UnitModeCurrent = E_UnitMode.Auto THEN
	GVL_ADS.MachineMode.CurrentMode := E_MachineMode.AUTO;
END_IF

ACTION A00_BasicUnit:
CoreSys_Start := MachineControl.Machine_Start;
CoreSys_Stop := MachineControl.Machine_Stop;
CoreSys_Reset := MachineControl.Machine_Reset;
MachineControl(
    eModeCommand := PackTags[0].Command.UnitMode,
    eStateCommand := PackTags[0].Command.CntrlCmd,
    PackTag := PackTags[0],
    INPUT := GVL_Input.uniDI.stDI,
    OUTPUT := GVL_Output.uniDO.stDO); // FB_MachineControl
PackTags[0].Status.StateCurrent := MachineControl.eStateCurrent;
PackTags[0].Status.UnitModeCurrent := MachineControl.eModeCurrent;
CoreSys_Estop := MachineControl.Machine_Estop;
END_ACTION

ACTION A01_UnitModeConfig:
//UserModeCofig(
//	eMode							:= ePMLUnitMode_Service, 
//	bDisableClearing				:= TRUE, 
//	bDisableStarting				:= TRUE, 
//	bDisableSuspended				:= FALSE, 
//	bDisableStopping				:= TRUE, 
//	bDisableAborting				:= TRUE, 
//	bDisableHolding					:= TRUE, 
//	bDisableHeld					:= TRUE, 
//	bDisableUnholding				:= TRUE, 
//	bDisableSuspending				:= TRUE, 
//	bDisableUnsuspending			:= TRUE, 
//	bDisableResetting				:= TRUE, 
//	bDisableIdle					:= TRUE, 
//	bDisableCompleting				:= TRUE, 
//	bDisableComplete				:= TRUE, 
//	bEnableUnitModeChangeStopped	:= TRUE, 
//	bEnableUnitModeChangeIdle		:= FALSE, 
//	bEnableUnitModeChangeSuspended	:= FALSE, 
//	bEnableUnitModeChangeExecute	:= FALSE, 
//	bEnableUnitModeChangeAborted	:= TRUE, 
//	bEnableUnitModeChangeHeld		:= FALSE, 
//	bEnableUnitModeChangeComplete	:= FALSE, 
//	bError							=> , 
//	nErrorId						=> );
END_ACTION

ACTION A10_StatusCtrl:
IF PackTags[0].Status.UnitModeCurrent = E_UnitMode.Manual THEN
	IF PackTags[0].Status.StateCurrent = ePMLState_Aborted AND NOT MachineControl.Error THEN
		PackTags[0].Command.CntrlCmd := ePMLCommand_Clear;
	END_IF
	IF PackTags[0].Status.StateCurrent = ePMLState_Stopped THEN
		IF OP_Mode = E_UnitMode.Manual THEN
		PackTags[0].Command.CntrlCmd := ePMLCommand_Reset;
		END_IF
	END_IF
	IF PackTags[0].Status.StateCurrent = ePMLState_Idle THEN
		PackTags[0].Command.CntrlCmd := ePMLCommand_Start;
	END_IF
ELSIF PackTags[0].Status.UnitModeCurrent = E_UnitMode.Auto THEN
	IF PackTags[0].Status.StateCurrent = ePMLState_Aborted AND NOT MachineControl.Error THEN
		PackTags[0].Command.CntrlCmd := ePMLCommand_Clear;
	END_IF
	IF PackTags[0].Status.StateCurrent = ePMLState_Stopped THEN
		IF OP_Mode = E_UnitMode.Auto THEN
		PackTags[0].Command.CntrlCmd := ePMLCommand_Reset;
		END_IF
	END_IF
	IF PackTags[0].Status.StateCurrent = ePMLState_Idle THEN
		PackTags[0].Command.CntrlCmd := ePMLCommand_Start;
	END_IF
END_IF

IF PackTags[0].Status.UnitModeCurrent = E_UnitMode.Manual THEN
    IF ((PackTags[0].Status.StateCurrent = ePMLState_Stopped) OR
        (PackTags[0].Status.StateCurrent = ePMLState_Aborted) OR
        (PackTags[0].Status.StateCurrent = ePMLState_Execute)) AND
        MachineControl.MachineHomed
        THEN
        IF OP_Mode = E_UnitMode.Auto THEN
            PackTags[0].Command.UnitMode := E_UnitMode.Auto;
			IF PackTags[0].Status.StateCurrent = ePMLState_Execute THEN
				PackTags[0].Command.CntrlCmd := ePMLCommand_Stop;
			END_IF
        END_IF
    END_IF
ELSIF PackTags[0].Status.UnitModeCurrent = E_UnitMode.Auto THEN
    IF ((PackTags[0].Status.StateCurrent = ePMLState_Stopped) OR
        (PackTags[0].Status.StateCurrent = ePMLState_Aborted) OR
        (PackTags[0].Status.StateCurrent = ePMLState_Execute))
        THEN
        IF OP_Mode = E_UnitMode.Manual THEN
			IF PackTags[0].Status.StateCurrent <> ePMLState_Aborted OR PackTags[0].Status.StateCurrent <> ePMLState_Aborting THEN
				PackTags[0].Command.CntrlCmd := ePMLCommand_Abort;
			END_IF
            PackTags[0].Command.UnitMode := E_UnitMode.Manual;
        END_IF
    END_IF
END_IF

//GVL_ADS.OpPannel_Status.EStopBtnStatus := CoreSys_Estop;
//GVL_ADS.OpPannel_Status.ResetBtnStatus := CoreSys_Reset;
//GVL_ADS.OpPannel_Status.StartBtnStatus := CoreSys_Start;
//GVL_ADS.OpPannel_Status.StopBtnStatus := CoreSys_Stop;
// Start
IF PackTags[0].Status.UnitModeCurrent = E_UnitMode.Auto THEN
	CASE PackTags[0].Status.StateCurrent OF
		ePMLState_Idle:
			IF CoreSys_Start THEN
				PackTags[0].Command.CntrlCmd := ePMLCommand_Start;
			END_IF
	END_CASE
END_IF

// Reset & Clear

IF PackTags[0].Status.UnitModeCurrent = E_UnitMode.Auto THEN
	CASE PackTags[0].Status.StateCurrent OF
		ePMLState_Stopped,ePMLState_Complete:
			IF CoreSys_Reset THEN
				PackTags[0].Command.CntrlCmd := ePMLCommand_Reset;
			END_IF
		ePMLState_Aborted:
			IF CoreSys_Reset THEN
				PackTags[0].Command.CntrlCmd := ePMLCommand_Clear;
			END_IF
		ePMLState_Held:
			IF CoreSys_Reset THEN
				PackTags[0].Command.CntrlCmd := ePMLCommand_Unhold;
			END_IF
		ePMLState_Suspended:
			IF CoreSys_Reset THEN
				PackTags[0].Command.CntrlCmd := ePMLCommand_Unsuspend;
			END_IF
	END_CASE
END_IF

// === 光電板斷點重啟 ===
// 按 Reset 時若有 851~854 alarm,順便 power cycle Y10.5/Y10.6,
// 合併到既有 Reset 流程,不用操作員另外去找 Reboot Modbus 按鈕。
// R_TRIG 抓上升緣 + Status.Busy 雙重保險避免連續觸發。
trigResetForRS485(CLK := CoreSys_Reset);
IF trigResetForRS485.Q AND
   (   (MAIN2_RS485.RS485_V2[1].bError AND NOT GVL_HMI.Setup.Mechanical.stModbusByPass.switchOff_1)
    OR (MAIN2_RS485.RS485_V2[2].bError AND NOT GVL_HMI.Setup.Mechanical.stModbusByPass.switchOff_2)
    OR (MAIN2_RS485.RS485_V2[3].bError AND NOT GVL_HMI.Setup.Mechanical.stModbusByPass.switchOff_3)
    OR (MAIN2_RS485.RS485_V2[4].bError AND NOT GVL_HMI.Setup.Mechanical.stModbusByPass.switchOff_4))
   AND NOT GVL_ADS.RebootModbusDevices.Status.Busy
THEN
    GVL_ADS.RebootModbusDevices.Command.Execute := TRUE;
END_IF

// reboot 完成自動清 Execute,讓下次 Reset 還能觸發
IF GVL_ADS.RebootModbusDevices.Status.Done THEN
    GVL_ADS.RebootModbusDevices.Command.Execute := FALSE;
END_IF

 //Stop

IF PackTags[0].Status.UnitModeCurrent = E_UnitMode.Auto THEN
	CASE PackTags[0].Status.StateCurrent OF
		ePMLState_Execute:
			IF CoreSys_Stop THEN
				PackTags[0].Command.CntrlCmd := ePMLCommand_Suspend;
			END_IF
	END_CASE
END_IF
END_ACTION

END_PROGRAM

// ---- Library/20_MachineUnits/22_AllocateArea/Service/FB_AllocateMoveAutoBatchMode_Reverse.TcPOU
FUNCTION_BLOCK FB_AllocateMoveAutoBatchMode_Reverse EXTENDS FB_ObjectBase_V2
VAR_INPUT
//    Execute    :BOOL;   // True : This prog will start.
//    Abort      :BOOL;   // True : This prog will be abort.
//    Reset      :BOOL;   // True : This prog will be reset.
//    ObjectName :STRING; // Set this fb name(About it's action)
//	  Pause		 :BOOL;
	bOccupied							: BOOL;	
	Clips 								: REFERENCE TO  ARRAY[0..3] OF FB_Cylinder;
	cylinders 							: REFERENCE TO  ARRAY[0..3] OF FB_Cylinder;	
	TurnTable_Press		 		   		: REFERENCE TO FB_Cylinder;
	RoundBelt_Press 			   		: REFERENCE TO FB_Cylinder;
	AutoAllocateJobBatch_Reverse_Ctrl   :st_AllocateMoveAutoBatchMode_Ctrl;
	INPUT            			   		: REFERENCE TO ST_InputTable;
    OUTPUT           			   		: REFERENCE TO ST_OutputTable;
	NrOfAllocateCylinder 		   		: INT :=4;
	CurrentData 				   		: REFERENCE TO ST_SetupPara; // Componets setup parameter
	bAutoAllocateJobDryRun         		: BOOL := FALSE;
	RoundBeltMoveJob_Status 			: ST_StatusBasic;
END_VAR

VAR_OUTPUT
//    Busy    :BOOL;        // True : This prog is running.
//    Done    :BOOL;        // True : Command has been executed.
//    Aborted :BOOL;        // True : This prog is aborted.
//    Error   :BOOL;        // True : This prog has an error.
//    ErrorID :UINT;       // Output ErrorID
//    Status  :T_MaxString; // Output this prog status by string(255bytes)
	RoundBeltMoveJob_Ctrl : ST_CommandBasic;
	ProcessedIndex : ARRAY[0..49] OF INT;
	//UniqueErrorCode :STRING;
	// AutoAllocateJobBatch_Status    :st_AllocateMoveAutoBatchMode_Status;
	RoundBeltMoveJob_Position	:LREAL;
	bAllocateRobotMoveRequest : BOOL;
END_VAR

VAR
//    eState :E_MethodStatus_Basic;
//	uiExecutingStep : UDINT; // This var is used to been controll STATE_EXECUTING process.
//	uiResettingStep : UDINT;
//	uiAbortingStep : UDINT;
//	_Executed :BOOL; // Executing process completed.
//	_Error : BOOL; // FB has an error.
//	_ResetCompleted : BOOL; // FB resetting completed.
//	_AbortCompleted : BOOL; // FB aborting completed.
//	_Abort		: BOOL;
	strStatus	: STRING;
	uiResumeStep : UINT;

//	bSimpleAllocationBatchEnable		 :BOOL;
//	AutoRotatebelt_Internal_Ctrl   : st_RoundBeltAutoSingleMove_Ctrl;
	_UniqueErrorCode : STRING;
	arrProcessedIndex : ARRAY[0..49] OF INT;
 //   eState              :E_MethodStatus_Basic;  
  //  uiAbortingStep      :UDINT;
    uiAbortedStep       :UDINT;
  //  uiResettingStep     :UDINT;
	uiResumableStep		: E_AllocationJob;
    bAborttingCompleted :BOOL; // True: Aborting process finished
    bAborted            :BOOL; // True : Aborted process finished
    bExecuted           :BOOL; // True : Executing process finished
    bResettingCompleted :BOOL; // True : Resetting process finished  
    iWorkingIndex		:UINT:=0;	
	iProcessingIndex	:INT :=0;
	iWorkingCylinder	:INT;
	//_Error				:BOOL :=FALSE;
	StatusDescription	:STRING;
	ClipsHaveNeedle		: ARRAY[0..3] OF BOOL;
	ClipsHaveNeedle_Pick		: ARRAY[0..3] OF BOOL;
	ClipsHaveNoNeedle	: ARRAY[0..3] OF BOOL;
	bCylinderCheck 		: BOOL;
	bCylinderCheckFastMode : BOOL;
	iPickingNeedleCount		:INT;
	iPlacingNeedleCount		:INT;
	bIfNextCycle			:BOOL;
	bCheckStation			:BOOL:=FALSE;
	
	
	
	tAutoAllocationJobBatchTimeOut_Reverse:Tc2_Standard.TON;
    sAllocationJobBatchStatus      :STRING;
    tonFastModeTimeDelayBatch_Reverse      :Tc2_Standard.TON;
	AllocationJobBatchModeReverse		:E_AllocationJob := E_AllocationJob.Defult;
	 Ton_RoundBeltArrivedDelay     : TON;
	 CurrentPosition : ST_PositionTable;
	
  	RoundBeltMoveJob : st_AllocateCircleMoveStructure;	
		
//==========================M_AllocationJobBatchMode================================

	{attribute 'hide'}
	bCheckTrue : BOOL:=TRUE;
	iCurrentRotateBeltStation : UINT;
	i : UINT;	
	j : UINT;	

	bMoveRotateBeltBusy	:BOOL;
	bMoveRotateBeltDone : BOOL;
	A1Used				:BOOL :=FALSE;
	A2Used				:BOOL :=FALSE;
	R1Used				:BOOL :=FALSE;
	R2Used				:BOOL :=FALSE;
	bBoxCheck			:BOOL :=TRUE;
	PickingStation		:UINT;
	iNextPickingStation :UINT;
	
	_bRetry : BOOL;

	
	
END_VAR

A00_BasicUnits();
SUPER^.A10_StateControl();

(*============================================================
Create Date : 2026/04/27	
Last Update	: 2026/04/27
Change Log  : 導入鏡射機測試完成版本。 edited by Gamin 
============================================================*)

ACTION A00_BasicUnits:
Ton_RoundBeltArrivedDelay();
tonFastModeTimeDelayBatch_Reverse(PT:=T#100MS);
// 暫停時重置 Timeout 計時器，避免續作誤報超時
IF Pause THEN
    tAutoAllocationJobBatchTimeOut_Reverse.IN := FALSE;
END_IF
tAutoAllocationJobBatchTimeOut_Reverse(PT:=T#120s);	// 原 30s 太短,belt 移動 + XY 到位經常超時
END_ACTION

METHOD GetModelState
VAR_OUTPUT
    xDone    :BOOL;
    xBusy    :BOOL;
    xError   :BOOL;
    xAborted :BOOL;
    iErrorID :UDINT;
	UniqueErrorCode : STRING;
END_VAR
xDone    := Done;
xBusy    := Busy;
xError   := Error;
xAborted := Abort;
iErrorID := ErrorID;
END_METHOD

METHOD GetName : STRING
GetName := ObjectName;
END_METHOD

(* Check Allocate Robot Clip cylinder no error
	Return True : no error
*)
METHOD M_CheckClipsNoError : BOOL
VAR_INPUT
END_VAR
//IF Clips[E_ClipsNo.ClipA].bError OR Clips[E_ClipsNo.ClipB].bError OR Clips[E_ClipsNo.ClipC].bError OR Clips[E_ClipsNo.ClipD].bError THEN
//    M_CheckClipsNoError := FALSE;
//ELSE
//    M_CheckClipsNoError := TRUE;
//END_IF
M_CheckClipsNoError := TRUE;
END_METHOD

(* Check Allocate Robot vertical cylinder no error
	return True : no error
*)
METHOD M_CheckCylindersNoError : BOOL
VAR_INPUT
END_VAR
//IF cylinders[E_CylinderNo.CylinderA].bError OR
//   cylinders[E_CylinderNo.CylinderB].bError OR
//   cylinders[E_CylinderNo.CylinderC].bError OR
//   cylinders[E_CylinderNo.CylinderD].bError
//THEN
//    M_CheckCylindersNoError := FALSE;
//ELSE
//    M_CheckCylindersNoError := TRUE;
//END_IF

M_CheckCylindersNoError := TRUE;
END_METHOD

METHOD PRIVATE M_RecoveryAxes : BOOL
VAR_INPUT
END_VAR
VAR
	bCheckTrue : BOOL;
	CheckErrorIndex : UINT;
END_VAR
bCheckTrue := TRUE;
FOR CheckErrorIndex:=1 TO 4 DO 
	IF arAxisCtrl_gb[CheckErrorIndex].Admin.Axis.Status.Error THEN
		arAxisCtrl_gb[CheckErrorIndex].Admin.ClearError:=TRUE;
		bCheckTrue:=FALSE;
	ELSE
		arAxisCtrl_gb[CheckErrorIndex].Admin.ClearError:=FALSE;
	END_IF
END_FOR
//		TurnTable := 1,
//      RoundBelt := 2,
//      Allocate_X := 3,
//      Allocate_Y := 4,

M_RecoveryAxes:= bCheckTrue;
END_METHOD

METHOD  M_STATE_ABORTED
VAR_INPUT
END_VAR
IF NOT _bRetry THEN
	Busy    := FALSE;
	Aborted := TRUE;
	Status  := StatusDescription;
	Error   := TRUE;
	uiAbortingStep:=0;
	_AbortCompleted := FALSE;
	ErrorID := GVL_ErrorCode.GC_SVCID_ALC_BATCH_FULL;
END_IF

IF reset THEN
	Aborted := FALSE;
	Error	:= FALSE;
	_bRetry := TRUE;
END_IF

IF NOT Execute THEN
    eState := STATE_RESETTING;
ELSIF Execute AND _bRetry THEN
	AllocationJobBatchModeReverse :=uiResumableStep;
	_bRetry := FALSE;
	eState :=STATE_EXECUTING;
END_IF
END_METHOD

METHOD  M_STATE_ABORTING
VAR_INPUT
END_VAR
CASE uiAbortingStep OF
		0:
			_Abort  := FALSE;
			_bRetry := FALSE;
			tAutoAllocationJobBatchTimeOut_Reverse.IN:=FALSE;
			Ton_RoundBeltArrivedDelay(IN := FALSE);
			RoundBeltMoveJob.HandShake.Execute := FALSE;
			RoundBeltMoveJob_Ctrl.Execute := FALSE;
			bAllocateRobotMoveRequest := FALSE;

			uiAbortingStep:=100;
			
		100:
			FOR i:=0 TO 3 DO
				IF cylinders[i].xError THEN
					cylinders[i].M_Reset();
				ELSE
					cylinders[i].M_Retract();	
				END_IF
			END_FOR
			uiAbortingStep:=9000;
				
		9000:
			_AbortCompleted := TRUE;
END_CASE

IF 	NOT Execute THEN
	eState := STATE_RESETTING;
ELSIF Execute AND _AbortCompleted THEN
	eState := STATE_Aborted;
END_IF
END_METHOD

METHOD  M_STATE_DONE
VAR_INPUT
END_VAR
Busy := FALSE;
Done := TRUE;
RoundBeltMoveJob.HandShake.Execute:=FALSE;
RoundBeltMoveJob_Ctrl.Execute:= RoundBeltMoveJob.HandShake.Execute;

DAS_CoreSys.MachineControl.fbAllocateArea.M_ReleaseRoundBeltAccess(E_RoundBeltControlAccess.Allocating);
IF Done AND NOT Execute THEN
    eState := STATE_DORMANT;
END_IF
END_METHOD

METHOD  M_STATE_DORMANT
VAR_INPUT
END_VAR
VAR
	_arrProcessedIndex : ARRAY[0..49] OF INT;	// 預設值全 0,用來清空 arrProcessedIndex / ProcessedIndex
END_VAR
Aborted         := FALSE;
Error           := FALSE;
ErrorID         := 0;
Busy                         := FALSE;
Done                         := FALSE;
_ResetCompleted := FALSE;
_Error          := FALSE;
_Executed       := FALSE;
_Abort			:= FALSE;
Aborted			:= FALSE;
strStatus := M_FormatManagedStatus(
	AlarmId := GVL_ErrorCode.GC_ALARM_ALC_BATCH_REVERSE,
	InnerMessage := GVL_ErrorCode.GC_MSG_0089);
Status := '';
Error := FALSE;
Status          := '';

uiExecutingStep :=uiResettingStep :=uiResumeStep :=0;
AllocationJobBatchModeReverse := E_AllocationJob.PreDataProcess;
i :=0;
j :=0;
iProcessingIndex :=0;
iWorkingCylinder :=0;
iWorkingIndex                := 0;	
Ton_RoundBeltArrivedDelay.IN := FALSE;
tAutoAllocationJobBatchTimeOut_Reverse.IN := FALSE;
bAllocateRobotMoveRequest	 := FALSE;

R1Used                       := FALSE;
R2Used                       := FALSE;
A1Used                       := FALSE;
A2Used                       := FALSE;
bMoveRotateBeltDone          := FALSE;	
bIfNextCycle				 := FALSE;	
bResettingCompleted :=FALSE;
ClipsHaveNeedle		:=
ClipsHaveNeedle_Pick:=
ClipsHaveNoNeedle	;
_bRetry := FALSE;

// 清空上一輪的 ProcessedIndex 回報,避免下一批次混到舊資料
// (對齊 FB_AllocateMoveAutoBatchMode 的作法: 用本地預設值 array 蓋掉)
arrProcessedIndex := _arrProcessedIndex;
ProcessedIndex    := _arrProcessedIndex;

IF Execute THEN

	eSTATE:=STATE_EXECUTING;
END_IF
END_METHOD

METHOD  M_STATE_ERROR
VAR_INPUT
END_VAR
Busy                         := FALSE;
Error                        := TRUE;
tAutoAllocationJobBatchTimeOut_Reverse.IN := FALSE;
Status                       := StatusDescription;
RoundBeltMoveJob.HandShake.Execute:=FALSE;
RoundBeltMoveJob_Ctrl.Execute:= RoundBeltMoveJob.HandShake.Execute;
DAS_CoreSys.MachineControl.fbAllocateArea.M_ReleaseRoundBeltAccess(E_RoundBeltControlAccess.Allocating);
FOR i:=0 TO 3 DO
	IF cylinders[i].xError THEN
		cylinders[i].M_Reset();
	ELSE
		cylinders[i].M_Retract();	
	END_IF
END_FOR

TurnTable_Press.M_Retract();
RoundBelt_Press.M_Retract();

IF NOT Execute THEN
    eState := STATE_RESETTING;
END_IF
END_METHOD

METHOD  M_STATE_EXECUTING
VAR_INPUT
END_VAR

VAR_INST
	CurrentProcessData	: ST_AllocationJobBatchModeInfo;
	CurrentPickingCoordinates : ARRAY[0..3] OF st_Coordinate;
	CurrentPlacingCoordinates : ARRAY[0..3] OF st_Coordinate;
	CurrentSyncGroupPicking		  : ARRAY[0..3] OF UINT :=[0,1,2,3];
	CurrentSyncGroupPiacing		  : ARRAY[0..3] OF UINT :=[0,1,2,3];
	iFirstWorkIndex		:UINT;
END_VAR

VAR
	emptyCoordinate		: ST_Coordinate;
	AllocateRobot: INT;
END_VAR
		Busy := TRUE;

		// Pause gate:
		// 停止本 Service 繼續派發新動作,並關閉 timeout 計時。
		// 不清除圓帶的命令跟取消移動命令，以防暫停的不步序是在等待到位或者完成，避免卡死。
		IF Pause THEN
			Paused := TRUE;
			StatusDescription := 'Allocate batch reverse paused';
			tAutoAllocationJobBatchTimeOut_Reverse.IN := FALSE;
			Ton_RoundBeltArrivedDelay(IN := FALSE);
//			RoundBeltMoveJob.HandShake.Execute := FALSE;
//			RoundBeltMoveJob_Ctrl.Execute := FALSE;
//			bAllocateRobotMoveRequest := FALSE;
			RETURN;
		END_IF
		Paused := FALSE;
			
		// 非自動模式直接中止 (避免軸控衝突)
		IF GVL_Machine.PackTags[UnitNo.Allocate].Status.UnitModeCurrent <> E_UnitMode.Auto THEN
			StatusDescription := 'FB_AllocateMoveAutoBatchMode_Reverse Not in Auto mode';
			_UniqueErrorCode := 'E_NOT_AUTO_MODE';
			_Error := TRUE;
		END_IF

		// 每 cycle 把內部 arrProcessedIndex 拷到 VAR_OUTPUT,讓上位/MachineControl 隨時看到目前已處理的 ID
		// (對齊 FB_AllocateMoveAutoBatchMode 的作法)
		ProcessedIndex := arrProcessedIndex;

		// ============================================================
		// TurnTable Interlock (Safety)
		// 拔針 pick 階段 (CylinderDown ~ CylinderUp) 期間, cylinders 伸到
		// TurnTable 盒上方, TurnTable 絕對不可轉動, 否則撞斷 cylinder/夾爪
		// ============================================================
		IF (AllocationJobBatchModeReverse = E_AllocationJob.CylinderDownPick
		 OR AllocationJobBatchModeReverse = E_AllocationJob.ClipColse
		 OR AllocationJobBatchModeReverse = E_AllocationJob.CylinderUpPick) THEN
			IF arAxisCtrl_gb[AxisNo.TurnTable].Admin.Axis.Status.Moving THEN
				StatusDescription := 'TurnTable interlock: must not move during pick';
				_UniqueErrorCode := 'E_TT_INTERLOCK';
				uiResumableStep := AllocationJobBatchModeReverse;
				_Abort := TRUE;
				RETURN;
			END_IF
		END_IF

		DAS_CoreSys.MachineControl.fbAllocateArea.M_GetRoundBeltAccess(E_RoundBeltControlAccess.Allocating);
		RoundBeltMoveJob_Ctrl.Execute:=RoundBeltMoveJob.HandShake.Execute;
		RoundBeltMoveJob.HandShake.Busy:=RoundBeltMoveJob_Status.Busy;
		RoundBeltMoveJob.HandShake.Done:=RoundBeltMoveJob_Status.Done;
		RoundBeltMoveJob.HandShake.Error:=RoundBeltMoveJob_Status.Error;
		RoundBeltMoveJob_Position:=RoundBeltMoveJob.Position;
		
		CASE AllocationJobBatchModeReverse OF
			E_AllocationJob.PreDataProcess :
				IF NOT Pause THEN // Pausing here waiting pause finish
					
					bCheckStation:=FALSE;
					//Get current allocation data
					FOR i:=iProcessingIndex TO 	AutoAllocateJobBatch_Reverse_Ctrl.AutoMode_AllocateMoveBatch.NrOfAllocationJob-1 BY 1  DO
						CurrentProcessData := 	AutoAllocateJobBatch_Reverse_Ctrl.AutoMode_AllocateMoveBatch.AllocationInfo[iProcessingIndex];
						
						FOR j:=0 TO 3 DO
							IF NOT (CurrentProcessData.PlacingNeedleInfo[j].Station=99) THEN
									bCheckStation:=TRUE; //Station = 99 means this job should be ignou , Therefor any station of job is "not" 99 , means this job should be process
								EXIT;
							END_IF						
						END_FOR
						
						IF bCheckStation THEN
								AllocationJobBatchModeReverse:=E_AllocationJob.Idle;
								EXIT;
							ELSE
								iProcessingIndex:=iProcessingIndex+1;
								arrProcessedIndex[i] :=CurrentProcessData.ID;
						END_IF						
					END_FOR		

					IF 		AutoAllocateJobBatch_Reverse_Ctrl.AutoMode_AllocateMoveBatch.NrOfAllocationJob<= iProcessingIndex THEN
							AllocationJobBatchModeReverse:=E_AllocationJob.Finish;
					END_IF				
				END_IF
				
		
		
		
		
		
			E_AllocationJob.Idle:
				//idle 
								
				FOR i:=0 TO 3 DO
					IF CurrentProcessData.PickingNeedleInfo[i].CycleStart THEN
						FUN_GetNeedleCoordinates(uiLocation:=1,
										uiBox:=CurrentProcessData.PickingNeedleInfo[i].Box,
										uiClip:=CurrentProcessData.PickingNeedleInfo[i].Clip,
										uiNeedleLocation :=CurrentProcessData.PickingNeedleInfo[i].NeedleLocation,
										NeedleCoordinate=>CurrentPickingCoordinates[i]);
				
						CurrentSyncGroupPicking[i] :=i;
					ELSE
						CurrentPickingCoordinates[i]:=	emptyCoordinate;
						CurrentSyncGroupPicking[i] :=99;
					END_IF
					
					IF CurrentProcessData.PlacingNeedleInfo[i].CycleStart THEN
						FUN_GetNeedleCoordinates(uiLocation:=0,
										uiBox:=CurrentProcessData.PlacingNeedleInfo[i].Box,
										uiClip:=CurrentProcessData.PlacingNeedleInfo[i].Clip,
										uiNeedleLocation :=CurrentProcessData.PlacingNeedleInfo[i].NeedleLocation,
										NeedleCoordinate=>CurrentPlacingCoordinates[i]);
						CurrentSyncGroupPiacing[i] :=i;				
					ELSE
							CurrentPlacingCoordinates[i]:=	emptyCoordinate;
							CurrentSyncGroupPiacing[i] :=99;	
					END_IF
									
												
				
				
					ClipsHaveNeedle_Pick[i]:=CurrentProcessData.PickingNeedleInfo[i].CycleStart;
					ClipsHaveNeedle[i]	   :=CurrentProcessData.PlacingNeedleInfo[i].CycleStart;
					//Get placing needle info	
				END_FOR
				
				FUN_GetSyncGroup_AllocationJob(Coordinates :=CurrentPickingCoordinates,NeedleInfo:=CurrentProcessData.PickingNeedleInfo, SyncGroup=>CurrentSyncGroupPicking);
				FUN_GetSyncGroup_AllocationJob(Coordinates :=CurrentPlacingCoordinates,NeedleInfo:=CurrentProcessData.PlacingNeedleInfo, SyncGroup=>CurrentSyncGroupPiacing);	
				
				//Copy needle info to placing info
				tAutoAllocationJobBatchTimeOut_Reverse.IN:=FALSE;
				
				AllocationJobBatchModeReverse:=E_AllocationJob.Initial;
	
			E_AllocationJob.Initial:						
				//Get All cylinders & clips back
				bCheckTrue:=TRUE;
				
				tAutoAllocationJobBatchTimeOut_Reverse.IN:=TRUE	;
				
				FOR i:=0 TO NrOfAllocateCylinder-1 DO
					clips[i].M_Retract();//('E_AllocationJob.Initial');
					IF  clips[i].InRearPosition THEN
						cylinders[i].M_Retract();//('E_AllocationJob.Initial');
					END_IF

					IF NOT cylinders[i].InRearPosition THEN
						bCheckTrue:=FALSE;
					END_IF

				END_FOR
//					IF TurnTable.Motor.Error THEN
//					TurnTable.Motor.Reset();
//					bCheckTrue:=FALSE;
//				END_IF
				
//				IF  AllocateRobot.axX.Error THEN
//					  AllocateRobot.axX.Reset();
//					  bCheckTrue:=FALSE;
//				END_IF
				
//				IF  AllocateRobot.axY.Error THEN
//					  AllocateRobot.axY.Reset();
//					  bCheckTrue:=FALSE;
//				END_IF
				
//				IF RoundBelt.Motor.Error THEN
//					RoundBelt.Motor.Reset();
//				    bCheckTrue:=FALSE;				
//				END_IF
				
				IF bCheckTrue THEN	
					tAutoAllocationJobBatchTimeOut_Reverse.IN:=FALSE	;	
					IF bAutoAllocateJobDryRun THEN
						// Dry run mode will not check if boxes is ready						
						AllocationJobBatchModeReverse:=E_AllocationJob.MoveToTargetPos;
					ELSE						
						AllocationJobBatchModeReverse:=E_AllocationJob.CheckBoxesOnTurnTableReady;
					END_IF
					
				END_IF
				IF tAutoAllocationJobBatchTimeOut_Reverse.Q THEN
					StatusDescription :='initiial Cylindes timeout';
					uiResumableStep := E_AllocationJob.Initial;
					_Abort :=TRUE;					
				END_IF
	
	E_AllocationJob.CheckBoxesOnTurnTableReady:
		//Check box is ready on turntable
		// TurnTable 角度 gate: 必須在 0/90/180/270 (任一 station) 才允許拔針
		// 取絕對值處理負角度 (e.g., -90 → 90, -180 → 180)
		IF NOT (FUN_CheckInPos(ActPos:=ABS(arAxisCtrl_gb[AxisNo.TurnTable].Admin.Axis.NcToPlc.ModuloActPos), TargetPos:=0,   ToleranceRange:=0.1)
		     OR FUN_CheckInPos(ActPos:=ABS(arAxisCtrl_gb[AxisNo.TurnTable].Admin.Axis.NcToPlc.ModuloActPos), TargetPos:=90,  ToleranceRange:=0.1)
		     OR FUN_CheckInPos(ActPos:=ABS(arAxisCtrl_gb[AxisNo.TurnTable].Admin.Axis.NcToPlc.ModuloActPos), TargetPos:=180, ToleranceRange:=0.1)
		     OR FUN_CheckInPos(ActPos:=ABS(arAxisCtrl_gb[AxisNo.TurnTable].Admin.Axis.NcToPlc.ModuloActPos), TargetPos:=270, ToleranceRange:=0.1)
		     OR FUN_CheckInPos(ActPos:=ABS(arAxisCtrl_gb[AxisNo.TurnTable].Admin.Axis.NcToPlc.ModuloActPos), TargetPos:=360, ToleranceRange:=0.1)) THEN
			StatusDescription := 'TurnTable angle invalid: must be at 0/90/180/270 to pick';
			_UniqueErrorCode := 'E_TT_ANGLE_INVALID';
			_Error := TRUE;
		END_IF
		tAutoAllocationJobBatchTimeOut_Reverse.IN:=TRUE	;
		R1Used := FALSE;
		R2Used := FALSE;
		bBoxCheck :=TRUE;		
				FOR i:=0 TO 3 DO
					IF CurrentProcessdata.PickingNeedleInfo[i].CycleStart OR CurrentProcessdata.PlacingNeedleInfo[i].CycleStart THEN
						IF CurrentProcessdata.PickingNeedleInfo[i].Box=0 THEN
							R1Used :=TRUE;
							END_IF
						
						 IF  CurrentProcessdata.PickingNeedleInfo[i].Box=1 THEN
 							R2Used :=TRUE;
						END_IF
					END_IF
				END_FOR
				
				IF  R1Used THEN 
					  bBoxCheck :=INPUT.bTurnTable_I1Detect_Sensor AND bBoxCheck; 
				END_IF
				IF  R2Used THEN 
					  bBoxCheck :=INPUT.bTurnTable_I2Detect_Sensor AND bBoxCheck; 
				END_IF
 				
				IF bBoxCheck THEN
						bBoxCheck:=FALSE;
						IF NOT TurnTable_Press.InFrontPosition THEN
							TurnTable_Press.M_Extend();// .M_Extend();//('Auto Mode Allocation Batch Mode reverse : Turn table press box Forward');
						END_IF
						AllocationJobBatchModeReverse:=E_AllocationJob.MoveToTargetPos;
				END_IF
				
				IF tAutoAllocationJobBatchTimeOut_Reverse.Q THEN
					uiResumableStep := E_AllocationJob.CheckBoxesOnTurnTableReady;
					_Abort :=TRUE	;
					StatusDescription :='Box not ready on Turn table';
				END_IF
				
	E_AllocationJob.MoveToTargetPos:
				// Move to picking position
                Ton_RoundBeltArrivedDelay(IN := FALSE);
                tAutoAllocationJobBatchTimeOut_Reverse.IN := FALSE;

				IF ClipsHaveNeedle_Pick[iWorkingIndex] THEN // Work if this index is request
                	iWorkingCylinder := CurrentProcessData.PickingNeedleInfo[iWorkingIndex].Clip;
					// Get working cylinder index from picking info
					IF cylinders[iWorkingCylinder].InRearPosition THEN
					bAllocateRobotMoveRequest	:= TRUE;		
						// Move allocating robot to picking position
					arAxisCtrl_gb[AxisNo.Allocate_X].PosMode.Acc := CurrentData.Axes.Allocate_X.HalfAuto.Acceleration;
					arAxisCtrl_gb[AxisNo.Allocate_X].PosMode.Dec := CurrentData.Axes.Allocate_X.HalfAuto.Deceleration;
					arAxisCtrl_gb[AxisNo.Allocate_X].PosMode.Jerk := CurrentData.Axes.Allocate_X.HalfAuto.Jerk;
					arAxisCtrl_gb[AxisNo.Allocate_X].PosMode.Velocity := CurrentData.Axes.Allocate_X.HalfAuto.Velocity;
					arAxisCtrl_gb[AxisNo.Allocate_X].PosMode.Position :=CurrentPickingCoordinates[iWorkingIndex].X;

					arAxisCtrl_gb[AxisNo.Allocate_Y].PosMode.Acc := CurrentData.Axes.Allocate_Y.HalfAuto.Acceleration;
					arAxisCtrl_gb[AxisNo.Allocate_Y].PosMode.Dec := CurrentData.Axes.Allocate_Y.HalfAuto.Deceleration;
					arAxisCtrl_gb[AxisNo.Allocate_Y].PosMode.Jerk := CurrentData.Axes.Allocate_Y.HalfAuto.Jerk;
					arAxisCtrl_gb[AxisNo.Allocate_Y].PosMode.Velocity := CurrentData.Axes.Allocate_Y.HalfAuto.Velocity;
					arAxisCtrl_gb[AxisNo.Allocate_Y].PosMode.Position := CurrentPickingCoordinates[iWorkingIndex].Y;
					END_IF

              		FOR i :=0 TO 3 DO
						IF  CurrentProcessData.PlacingNeedleInfo[i].CycleStart THEN
							iFirstWorkIndex:=	i;
							EXIT;
							//Get the first working index in oreder to move the rotatebelt in Fast mode
						END_IF
					END_FOR
				

					IF CurrentProcessData.FastMode THEN //In Fast mode , RotateTable can start move at same moment 
						
		
					//	IF iCurrentRotateBeltStation <> CurrentProcessData.PlacingNeedleInfo[iFirstWorkIndex].Station THEN
							 //request to get the access to control Rotate belt
							RoundBeltMoveJob.Position:=CurrentProcessData.PlacingNeedleInfo[iFirstWorkIndex].Station;							
							RoundBeltMoveJob.HandShake.Execute;			
							// In fast mode , just send rotatebelt to target station if it's request different station. Station check will be later
					//	END_IF
				
					END_IF
						AllocationJobBatchModeReverse:=E_AllocationJob.MovingToTargetPos;		
//    	            IF AllocateRobot.P_isMoving   THEN
						
//        	            AllocationJobBatchModeReverse := E_AllocationJob.MovingToTargetPos;					 
					
//					ELSIF	 NOT AllocateRobot.P_isMoving AND_THEN  AllocateRobot.P_InTargetPosition THEN
//						AllocationJobBatchModeReverse := E_AllocationJob.MovingToTargetPos;	
//            	    END_IF
				
				ELSE
					AllocationJobBatchModeReverse:=E_AllocationJob.IfNextPTP_Picking;	
				END_IF

     E_AllocationJob.MovingToTargetPos:

                tAutoAllocationJobBatchTimeOut_Reverse.IN := TRUE;

//                IF AllocateRobot.P_InTargetPosition THEN
//                    tAutoAllocationJobBatchTimeOut_Reverse.IN := FALSE;
//                    tAutoAllocationJobBatchTimeOut_Reverse.PT := GVL.tAutoAllocateJobCylinderTimeout;
					
//				    AllocationJobBatchModeReverse                := E_AllocationJob.CylinderDownPick;
					
//                END_IF

				IF arAxisStatus_gb[AxisNo.Allocate_X].Admin.CmdDone AND arAxisStatus_gb[AxisNo.Allocate_Y].Admin.CmdDone 
					AND arAxisStatus_gb[AxisNo.Allocate_X].Admin._OpModeAck = ModePosAbs AND arAxisStatus_gb[AxisNo.Allocate_Y].Admin._OpModeAck = ModePosAbs THEN
					bAllocateRobotMoveRequest		:= FALSE;
					AllocationJobBatchModeReverse   := E_AllocationJob.CylinderDownPick;
				END_IF
                IF tAutoAllocationJobBatchTimeOut_Reverse.Q THEN
                    StatusDescription := 'Moving to picking position timeout';
                    _Abort            := TRUE;
					uiResumableStep	  :=E_AllocationJob.MoveToTargetPos;

                END_IF
				
	

            
	   E_AllocationJob.CylinderDownPick:
	   			// Cylinder move down to pick needle
                tAutoAllocationJobBatchTimeOut_Reverse.IN := TRUE;
				bCylinderCheck:=TRUE;                
                
                THIS^.cylinders[iWorkingCylinder].M_Extend();// //('AutoMode E_AllocationJob.CylinderDownPick');
				// Cylinder move down
				IF CurrentProcessData.SyncMode THEN //In sync mode , the cylinders in same sync group can move down at same step 
					FOR i := iWorkingIndex+1 TO 3 DO
						IF CurrentSyncGroupPicking[i]=CurrentSyncGroupPicking[iWorkingIndex] AND 
							ClipsHaveNeedle_Pick[i]	 THEN
							cylinders[CurrentProcessData.PickingNeedleInfo[i].Clip ].M_Extend();//('Auto Mode E_AllocationJob.CylinderDownPick in Sync placing Mode');
							bCylinderCheck :=cylinders[CurrentProcessData.PickingNeedleInfo[i].Clip ].InFrontPosition AND bCylinderCheck;			
						END_IF
					END_FOR
					
				END_IF
                
				
				
                IF cylinders[iWorkingCylinder].InFrontPosition AND bCylinderCheck THEN
                    tAutoAllocationJobBatchTimeOut_Reverse.IN := FALSE;
                    AllocationJobBatchModeReverse                := E_AllocationJob.ClipColse;
                END_IF

                IF tAutoAllocationJobBatchTimeOut_Reverse.Q THEN
					uiResumableStep := E_AllocationJob.CylinderDownPick;                    
                    _Abort            := TRUE;
					StatusDescription := 'Picking down timeout';
                END_IF

            E_AllocationJob.ClipColse:
				// Close clip to pick needke
                Ton_RoundBeltArrivedDelay.IN := FALSE;
                tAutoAllocationJobBatchTimeOut_Reverse.IN := TRUE;
				bCylinderCheck:=TRUE;
				
                THIS^.clips[iWorkingCylinder].M_Extend();//('Auto Mode E_AllocationJob.ClipColse');
						// Close clip
				IF CurrentProcessData.SyncMode THEN // In sync mode, the clips in same sync group can move together
					FOR i := iWorkingIndex+1 TO 3 DO
						IF CurrentSyncGroupPicking[i]=CurrentSyncGroupPicking[iWorkingIndex] AND 
							ClipsHaveNeedle_Pick[i]	 THEN
							clips[CurrentProcessData.PickingNeedleInfo[i].Clip ].M_Extend();//('Auto Mode E_AllocationJob.ClipColse in Sync placing Mode');
							bCylinderCheck :=clips[CurrentProcessData.PickingNeedleInfo[i].Clip ].InFrontPosition AND bCylinderCheck;			
						END_IF
					END_FOR
					
				END_IF
				
                IF clips[iWorkingCylinder].InFrontPosition AND bCylinderCheck THEN
                    tAutoAllocationJobBatchTimeOut_Reverse.IN := FALSE;
                    AllocationJobBatchModeReverse                := E_AllocationJob.CylinderUpPick;
                END_IF

                IF tAutoAllocationJobBatchTimeOut_Reverse.Q THEN

                    StatusDescription := 'Picking Close timeout, not can retry';
                    //uiResumableStep := E_AllocationJob.ClipColse;               // 如果夾盒不跳回上一步去做的話錯誤清理會縮回，會變成在上面夾
					//uiResumableStep := E_AllocationJob.CylinderDownPick;        // 不能續做 無法確保重新下去後是否有夾針。	
                    _Error            := TRUE;
                END_IF

	E_AllocationJob.CylinderUpPick:
		// Cylinder move up to pick needle
		bCylinderCheck:=TRUE;
		tAutoAllocationJobBatchTimeOut_Reverse.IN:=TRUE	;
		bBoxCheck:=TRUE;
			
		IF  R1Used THEN 
				  bBoxCheck :=INPUT.bTurnTable_I1Detect_Sensor  AND bBoxCheck; 
		END_IF
		IF  R2Used THEN 
				  bBoxCheck :=INPUT.bTurnTable_I2Detect_Sensor AND bBoxCheck; 
		END_IF
		
		THIS^.cylinders[iWorkingCylinder].M_Retract();//('Auto Mode E_AllocationJob.CylinderUpPick');		
	
		IF CurrentProcessData.SyncMode THEN
					FOR i := iWorkingIndex+1 TO 3 DO
						IF CurrentSyncGroupPicking[i]=CurrentSyncGroupPicking[iWorkingIndex] AND 
							ClipsHaveNeedle_Pick[i]	 THEN
							cylinders[CurrentProcessData.PickingNeedleInfo[i].Clip].M_Retract();//('Auto Mode E_AllocationJob.CylinderUpPick in Sync placing Mode');
							bCylinderCheck :=cylinders[CurrentProcessData.PickingNeedleInfo[i].Clip].InRearPosition AND bCylinderCheck;			
						END_IF
					END_FOR					
		END_IF
				
		IF cylinders[iWorkingCylinder].InRearPosition AND bCylinderCheck AND  bBoxCheck THEN
			R1Used:=FALSE;
			R2Used:=FALSE;
			tonFastModeTimeDelayBatch_Reverse.IN:=FALSE;		
			AllocationJobBatchModeReverse:=E_AllocationJob.IfNextPTP_Picking;
		END_IF
		
		IF tAutoAllocationJobBatchTimeOut_Reverse.Q THEN
			
			StatusDescription :='Picking Up timeout';
			uiResumableStep := E_AllocationJob.CylinderUpPick;                    
            _Abort            := TRUE;
		END_IF
		
	E_AllocationJob.IfNextPTP_Picking:
		// Check if next picking 
		iPickingNeedleCount:=1;
		IF CurrentProcessData.SyncMode THEN //Sync mode
			FOR i := iWorkingIndex+1 TO 3 DO
				IF CurrentSyncGroupPicking[i]=CurrentSyncGroupPicking[iWorkingIndex] AND 	ClipsHaveNeedle_Pick[i]	 THEN
					iPickingNeedleCount:=iPickingNeedleCount+1;
					ClipsHaveNeedle_Pick[i]:=FALSE;		
				END_IF
			END_FOR
		END_IF
		
		tAutoAllocationJobBatchTimeOut_Reverse.IN:=FALSE	;
		iWorkingIndex:=iWorkingIndex+1;
		IF iWorkingIndex>= NrOfAllocateCylinder THEN
			iWorkingIndex:=0;
			RoundBeltMoveJob.HandShake.Execute := FALSE;	// P1 fix: 改 HandShake (非 Ctrl),避免下 scan 被 line 429 覆蓋
			AllocationJobBatchModeReverse:=E_AllocationJob.CheckRotateBeltStation;	
			// If no more picking , go to next step to check  the rotate belt station 
		ELSE
			AllocationJobBatchModeReverse:=E_AllocationJob.MoveToTargetPos;
			// Still picking job , go back to next picking position
		END_IF
	
	
	E_AllocationJob.CheckRotateBeltStation:	
		// Check if the Rotate belt is in the target.
		
		IF ClipsHaveNeedle[iWorkingIndex] THEN
		
			tAutoAllocationJobBatchTimeOut_Reverse.IN:=FALSE;				
			iWorkingCylinder := CurrentProcessData.PlacingNeedleInfo[iWorkingIndex].Clip ;
			RoundBeltMoveJob.Position:=CurrentProcessData.PlacingNeedleInfo[iWorkingIndex].Station;			
			AllocationJobBatchModeReverse:=E_AllocationJob.MovingRotateBeltStation;				
		ELSE
				AllocationJobBatchModeReverse:=E_AllocationJob.IfNextPTP_Placing;	
		END_IF		
	
      E_AllocationJob.MovingRotateBeltStation:
				// timeout 保護: belt + XY 同時啟動,等兩者都就緒
				tAutoAllocationJobBatchTimeOut_Reverse.IN := TRUE;

                bMoveRotateBeltBusy := RoundBeltMoveJob_Status.Busy;
				bMoveRotateBeltDone := RoundBeltMoveJob_Status.Done;
                RoundBeltMoveJob.HandShake.Execute := TRUE;
				// XY 與圓帶同時啟動（不受 FastMode 限制）
				IF cylinders[iWorkingCylinder].InRearPosition THEN
					
					bAllocateRobotMoveRequest	:= TRUE;
					
					arAxisCtrl_gb[AxisNo.Allocate_X].PosMode.Acc := CurrentData.Axes.Allocate_X.HalfAuto.Acceleration;
					arAxisCtrl_gb[AxisNo.Allocate_X].PosMode.Dec := CurrentData.Axes.Allocate_X.HalfAuto.Deceleration;
					arAxisCtrl_gb[AxisNo.Allocate_X].PosMode.Jerk := CurrentData.Axes.Allocate_X.HalfAuto.Jerk;
					arAxisCtrl_gb[AxisNo.Allocate_X].PosMode.Velocity := CurrentData.Axes.Allocate_X.HalfAuto.Velocity;
					arAxisCtrl_gb[AxisNo.Allocate_X].PosMode.Position :=CurrentPlacingCoordinates[iWorkingIndex].X;

					arAxisCtrl_gb[AxisNo.Allocate_Y].PosMode.Acc := CurrentData.Axes.Allocate_Y.HalfAuto.Acceleration;
					arAxisCtrl_gb[AxisNo.Allocate_Y].PosMode.Dec := CurrentData.Axes.Allocate_Y.HalfAuto.Deceleration;
					arAxisCtrl_gb[AxisNo.Allocate_Y].PosMode.Jerk := CurrentData.Axes.Allocate_Y.HalfAuto.Jerk;
					arAxisCtrl_gb[AxisNo.Allocate_Y].PosMode.Velocity := CurrentData.Axes.Allocate_Y.HalfAuto.Velocity;
					arAxisCtrl_gb[AxisNo.Allocate_Y].PosMode.Position := CurrentPlacingCoordinates[iWorkingIndex].Y;
				END_IF
			
					
						
              	 IF (bMoveRotateBeltBusy OR bMoveRotateBeltDone) AND
				    (  arAxisCtrl_gb[AxisNo.Allocate_X].Admin.Axis.Status.Moving   OR arAxisCtrl_gb[AxisNo.Allocate_Y].Admin.Axis.Status.Moving
				    OR (arAxisStatus_gb[AxisNo.Allocate_X].Admin.CmdDone AND arAxisStatus_gb[AxisNo.Allocate_Y].Admin.CmdDone) )	 THEN
					tAutoAllocationJobBatchTimeOut_Reverse.IN := FALSE;
                 	   AllocationJobBatchModeReverse := E_AllocationJob.MovedRotateBeltStation;
               	 END_IF

				IF tAutoAllocationJobBatchTimeOut_Reverse.Q THEN
					StatusDescription := 'MovingRotateBeltStation: Belt or XY not responding timeout';
					uiResumableStep := E_AllocationJob.MovingRotateBeltStation;
					_Abort := TRUE;
				END_IF

      E_AllocationJob.MovedRotateBeltStation:

                tAutoAllocationJobBatchTimeOut_Reverse.IN := TRUE;

                bMoveRotateBeltDone := RoundBeltMoveJob_Status.Done;
                Ton_RoundBeltArrivedDelay(IN := bMoveRotateBeltDone);

                IF bMoveRotateBeltDone THEN
					RoundBeltMoveJob.HandShake.Execute := FALSE;  
					// XY 已在 MovingRotateBeltStation 啟動，直接等兩軸到位
					AllocationJobBatchModeReverse := E_AllocationJob.MovingToPlacingPos;
                END_IF
				
			 

                IF tAutoAllocationJobBatchTimeOut_Reverse.Q THEN
                    StatusDescription := 'Rotate Belt TimeOut';
					//uiResumableStep := E_AllocationJob.MovedRotateBeltStation;	這一步是在等done，如果回歸這一步仍不會叫圓帶移動。
					uiResumableStep := E_AllocationJob.MovingRotateBeltStation;
                    _Abort            := TRUE;	// P1 fix: 改 _Abort (可續做)
                END_IF

            E_AllocationJob.MoveToPlacingPos:

                IF ClipsHaveNeedle[iWorkingIndex] THEN
                    iWorkingCylinder := CurrentProcessData.PlacingNeedleInfo[iWorkingIndex].Clip;
					IF cylinders[iWorkingCylinder].InRearPosition THEN
						
						bAllocateRobotMoveRequest	:= TRUE;
						
						arAxisCtrl_gb[AxisNo.Allocate_X].PosMode.Acc := CurrentData.Axes.Allocate_X.HalfAuto.Acceleration;
						arAxisCtrl_gb[AxisNo.Allocate_X].PosMode.Dec := CurrentData.Axes.Allocate_X.HalfAuto.Deceleration;
						arAxisCtrl_gb[AxisNo.Allocate_X].PosMode.Jerk := CurrentData.Axes.Allocate_X.HalfAuto.Jerk;
						arAxisCtrl_gb[AxisNo.Allocate_X].PosMode.Velocity := CurrentData.Axes.Allocate_X.HalfAuto.Velocity;
						arAxisCtrl_gb[AxisNo.Allocate_X].PosMode.Position :=CurrentPlacingCoordinates[iWorkingIndex].X;
	
						arAxisCtrl_gb[AxisNo.Allocate_Y].PosMode.Acc := CurrentData.Axes.Allocate_Y.HalfAuto.Acceleration;
						arAxisCtrl_gb[AxisNo.Allocate_Y].PosMode.Dec := CurrentData.Axes.Allocate_Y.HalfAuto.Deceleration;
						arAxisCtrl_gb[AxisNo.Allocate_Y].PosMode.Jerk := CurrentData.Axes.Allocate_Y.HalfAuto.Jerk;
						arAxisCtrl_gb[AxisNo.Allocate_Y].PosMode.Velocity := CurrentData.Axes.Allocate_Y.HalfAuto.Velocity;
						arAxisCtrl_gb[AxisNo.Allocate_Y].PosMode.Position := CurrentPlacingCoordinates[iWorkingIndex].Y;

                        AllocationJobBatchModeReverse := E_AllocationJob.MovingToPlacingPos;
					END_IF                    

                ELSE

                    AllocationJobBatchModeReverse := E_AllocationJob.IfNextPTP_Placing;
                END_IF
				
	

            E_AllocationJob.MovingToPlacingPos:

                tAutoAllocationJobBatchTimeOut_Reverse.IN := TRUE;           		 
				IF arAxisStatus_gb[AxisNo.Allocate_X].Admin.CmdDone 
					AND arAxisStatus_gb[AxisNo.Allocate_Y].Admin.CmdDone
					AND arAxisStatus_gb[AxisNo.Allocate_X].Admin._OpModeAck = ModePosAbs
					AND arAxisStatus_gb[AxisNo.Allocate_Y].Admin._OpModeAck = ModePosAbs
					AND NOT arAxisCtrl_gb[AxisNo.RoundBelt].Admin.Axis.Status.Moving 
					AND  arAxisCtrl_gb[AxisNo.Allocate_X].Admin.Axis.Status.NotMoving
					AND  arAxisCtrl_gb[AxisNo.Allocate_Y].Admin.Axis.Status.NotMoving		THEN
					bAllocateRobotMoveRequest := FALSE;
					RoundBeltMoveJob.HandShake.Execute := FALSE; 
					tAutoAllocationJobBatchTimeOut_Reverse.IN := FALSE;
					IF RoundBelt_Press.InFrontPosition THEN // make sure press box cylinder is in front
							IF bAutoAllocateJobDryRun THEN
	                 		   AllocationJobBatchModeReverse                := E_AllocationJob.CylinderDownPlace;
							ELSE
								AllocationJobBatchModeReverse                := E_AllocationJob.CheckBoxReadyOnAllocatePosOfRoundBelt;
							END_IF
						ELSE
							RoundBelt_Press.M_Extend();//('');	
						END_IF
					
				END_IF
               

                IF tAutoAllocationJobBatchTimeOut_Reverse.Q THEN
                    StatusDescription := 'Moving placing timeout';
					//uiResumableStep := E_AllocationJob.MovingToPlacingPos;		//這一步是在等到位訊號，如果是回歸這一步仍不會動
					uiResumableStep := E_AllocationJob.MoveToPlacingPos;
                    _Abort            := TRUE;	// P1 fix: 改 _Abort (可續做),原本 _Error 不可續做
                END_IF

			E_AllocationJob.CheckBoxReadyOnAllocatePosOfRoundBelt:
				tAutoAllocationJobBatchTimeOut_Reverse.IN:=TRUE	;
				bBoxCheck := TRUE;		// P0 fix: 初始化,避免殘留 FALSE 導致永遠不進入
				A1Used := FALSE;		// P1 fix: resume 路徑殘留防呆
				A2Used := FALSE;

				  FOR i:=0 TO 3 DO
					IF CurrentProcessData.PlacingNeedleInfo[iWorkingIndex].Station = CurrentProcessData.PlacingNeedleInfo[i].Station THEN
						IF CurrentProcessData.PlacingNeedleInfo[i].Box=0 THEN
							A1Used :=TRUE;
							END_IF
						
					 	IF  CurrentProcessData.PlacingNeedleInfo[i].Box=1 THEN
 							A2Used :=TRUE;
						END_IF
					END_IF
				  END_FOR
				
				  IF  A1Used THEN 
					  bBoxCheck :=INPUT.bRoundBelt_WorkZoneQ1Detect_Sensor AND bBoxCheck; 
				  END_IF
				  IF  A2Used THEN 
					  bBoxCheck :=INPUT.bRoundBelt_WorkZoneQ2Detect_Sensor AND bBoxCheck; 
				  END_IF
 				
				  IF bBoxCheck THEN
						AllocationJobBatchModeReverse:=E_AllocationJob.CylinderDownPlace;
						A1Used := A2Used := FALSE;
				  END_IF
				
				IF tAutoAllocationJobBatchTimeOut_Reverse.Q THEN
					_Abort :=TRUE	;
					StatusDescription :='Box not ready on Rotate Belt';
					uiResumableStep := E_AllocationJob.CheckBoxReadyOnAllocatePosOfRoundBelt;
				END_IF	
				
            E_AllocationJob.CylinderDownPlace:
                bCylinderCheck               := TRUE;
                tAutoAllocationJobBatchTimeOut_Reverse.IN := TRUE;
                cylinders[iWorkingCylinder].M_Extend();//('Auto Mode E_AllocationJob.CylinderDownPlace');
				
				IF CurrentProcessData.SyncMode THEN
					FOR i := iWorkingIndex+1 TO 3 DO
						IF CurrentSyncGroupPiacing[i]=CurrentSyncGroupPiacing[iWorkingIndex] AND 
							ClipsHaveNeedle[i]	 THEN
							cylinders[CurrentProcessData.PlacingNeedleInfo[i].Clip].M_Extend();//('Auto Mode E_AllocationJob.CylinderDownPlace in Sync placing Mode');
							bCylinderCheck :=cylinders[CurrentProcessData.PlacingNeedleInfo[i].Clip].InFrontPosition AND bCylinderCheck;			
						END_IF
					END_FOR
					
				END_IF
				
               	 IF cylinders[iWorkingCylinder].InFrontPosition AND bCylinderCheck THEN
                    tAutoAllocationJobBatchTimeOut_Reverse.IN := FALSE;
                    AllocationJobBatchModeReverse                := E_AllocationJob.ClipOpen;
              	  END_IF
				
                IF tAutoAllocationJobBatchTimeOut_Reverse.Q THEN
                    StatusDescription := ' placing down timeout';
                    uiResumableStep := E_AllocationJob.CylinderDownPlace;                    
           			 _Abort            := TRUE;
                END_IF

            E_AllocationJob.ClipOpen:
                tAutoAllocationJobBatchTimeOut_Reverse.IN := TRUE;
                bCylinderCheck               := TRUE;
                clips[iWorkingCylinder].M_Retract();//('Auto Mode E_AllocationJob.ClipOpen');
					IF CurrentProcessData.SyncMode THEN
					FOR i := iWorkingIndex+1 TO 3 DO
						IF CurrentSyncGroupPiacing[i]=CurrentSyncGroupPiacing[iWorkingIndex] AND 
							ClipsHaveNeedle[i]	 THEN
							clips[CurrentProcessData.PlacingNeedleInfo[i].Clip].M_Retract();//('Auto Mode E_AllocationJob.ClipOpen in Sync placing Mode');
							bCylinderCheck :=clips[CurrentProcessData.PlacingNeedleInfo[i].Clip].InRearPosition AND bCylinderCheck;			
						END_IF
					END_FOR
					
				END_IF
				
				
                IF clips[iWorkingCylinder].InRearPosition AND bCylinderCheck THEN
                    tAutoAllocationJobBatchTimeOut_Reverse.IN := FALSE;
                    AllocationJobBatchModeReverse                := E_AllocationJob.CylinderUpPlace;
                END_IF

                IF tAutoAllocationJobBatchTimeOut_Reverse.Q THEN

                    StatusDescription := ' placing Close timeout, not can retry';
                   // uiResumableStep := E_AllocationJob.ClipOpen;  			// 如果回歸到這一步的話，報錯的時候汽缸會縮回，會導致在RearPos 就放掉
					//uiResumableStep := E_AllocationJob.CylinderDownPlace;     // 不能續做無法確定是否續做有風險             
           			 _Error            := TRUE;
                END_IF

            E_AllocationJob.CylinderUpPlace:
                bCylinderCheck         := TRUE;
				tAutoAllocationJobBatchTimeOut_Reverse.IN := TRUE;	// P0 fix: 原本沒啟動 timer → timeout 保護失效

                cylinders[iWorkingCylinder].M_Retract();//(' Auto Mode E_AllocationJob.CylinderUpPlace');

					IF CurrentProcessData.SyncMode THEN
					FOR i := iWorkingIndex+1 TO 3 DO
						IF CurrentSyncGroupPiacing[i]=CurrentSyncGroupPiacing[iWorkingIndex] AND
							ClipsHaveNeedle[i]	 THEN
							cylinders[CurrentProcessData.PlacingNeedleInfo[i].Clip].M_Retract();//('Auto Mode E_AllocationJob.CylinderUpPlace in Sync placing Mode');
							bCylinderCheck :=cylinders[CurrentProcessData.PlacingNeedleInfo[i].Clip].InRearPosition AND bCylinderCheck;

						END_IF
					END_FOR
				END_IF

                IF cylinders[iWorkingCylinder].InRearPosition AND bCylinderCheck THEN
                    tAutoAllocationJobBatchTimeOut_Reverse.IN              := FALSE;
                    AllocationJobBatchModeReverse := E_AllocationJob.CheckNeedlePlaced;

                END_IF

                IF tAutoAllocationJobBatchTimeOut_Reverse.Q THEN
                    StatusDescription := ' placing Up timeout';
                    uiResumableStep := E_AllocationJob.CylinderUpPlace;                    
           			 _Abort            := TRUE;
                END_IF

			E_AllocationJob.CheckNeedlePlaced: 
				ClipsHaveNeedle[iWorkingIndex] :=FALSE;
				IF CurrentProcessData.SyncMode THEN
					FOR i := iWorkingIndex+1 TO 3 DO
						IF CurrentSyncGroupPiacing[i]=CurrentSyncGroupPiacing[iWorkingIndex] AND ClipsHaveNeedle[i]	 THEN
							ClipsHaveNeedle[i]:=FALSE;
						END_IF
					END_FOR		
				END_IF
				AllocationJobBatchModeReverse := E_AllocationJob.IfNextPTP_Placing;
				
            E_AllocationJob.IfNextPTP_Placing:
                iWorkingIndex := iWorkingIndex + 1;

                IF iWorkingIndex >= NrOfAllocateCylinder THEN
                    iWorkingIndex := 0;
                    AllocationJobBatchModeReverse := E_AllocationJob.Finish;
                ELSE

                    AllocationJobBatchModeReverse := E_AllocationJob.CheckRotateBeltStation;
                END_IF

           
            E_AllocationJob.Finish:
                // Finish

               	arrProcessedIndex[iProcessingIndex] :=CurrentProcessData.ID;
				IF 	AutoAllocateJobBatch_Reverse_Ctrl.AutoMode_AllocateMoveBatch.NrOfAllocationJob> iProcessingIndex+1 THEN

					iProcessingIndex :=iProcessingIndex+1;
					AllocationJobBatchModeReverse := E_AllocationJob.PreDataProcess;
				ELSE
					// 最後一筆邏輯完成,但機械可能還在收尾。
					// 進入 FinalCleanup gate,等所有 cylinder/clip/press 都歸位、RoundBelt idle 才設 _Executed
					AllocationJobBatchModeReverse := E_AllocationJob.FinalCleanup;
				END_IF

			E_AllocationJob.FinalCleanup:
				// 給 Done 之前的最終收尾 gate:
				// 確保整批做完後,所有 cylinder/clip 都退到安全位置、RoundBelt 不再 Busy,
				// 才允許 _Executed := TRUE → STATE_DONE。
				// 目的: 上位看到 Done 時、PLC 內部資料(ProcessedIndex/WorkedID)跟機械都已穩定,
				//       上位撤 Execute 後即使馬上下一包進來也不會撞到上一包未收尾的狀態。
				// 註: TurnTable_Press / RoundBelt_Press 不收 — 兩個 Press 只是壓住盒子,
				//     對下一批的 X/Y robot 跟 cylinder 升降都沒有安全顧慮;
				//     收了反而會讓盒子晃動,且下一批 CheckBoxesOnTurnTableReady 還要再 Extend。
				tAutoAllocationJobBatchTimeOut_Reverse(IN := TRUE, PT := T#10S);
				bCheckTrue := TRUE;

				FOR i := 0 TO NrOfAllocateCylinder-1 DO
					clips[i].M_Retract();
					IF clips[i].InRearPosition THEN
						cylinders[i].M_Retract();
					END_IF
					IF NOT cylinders[i].InRearPosition OR NOT clips[i].InRearPosition THEN
						bCheckTrue := FALSE;
					END_IF
				END_FOR

				// 圓帶不可還在動作中
				IF RoundBeltMoveJob_Status.Busy THEN
					bCheckTrue := FALSE;
				END_IF

				// 同步把最後一筆 ID 確實出到 ProcessedIndex (頂部已每 cycle 拷貝,這裡是雙保險)
				ProcessedIndex := arrProcessedIndex;

				IF bCheckTrue THEN
					tAutoAllocationJobBatchTimeOut_Reverse.IN := FALSE;
					_Executed := TRUE;
				END_IF

				IF tAutoAllocationJobBatchTimeOut_Reverse.Q THEN
					StatusDescription := 'FinalCleanup timeout: hardware not back to safe position';
					_UniqueErrorCode := 'E_FINAL_CLEANUP_TIMEOUT';
					uiResumableStep := E_AllocationJob.FinalCleanup;
					_Abort := TRUE;
				END_IF
        END_CASE
			


	

IF NOT Execute THEN
	eState:=STATE_RESETTING;
END_IF
IF _Error THEN
	eState:=STATE_ERROR;
END_IF
IF _Abort THEN
	eSTATE:=STATE_ABORTING;
END_IF
IF _Executed THEN
	eSTATE:=STATE_Done;
END_IF
END_METHOD

METHOD  M_STATE_RESETTING
VAR_INPUT
END_VAR
Busy                         := FALSE;
Done                         := FALSE;
Error                        := FALSE;
_Error                       := FALSE;
tAutoAllocationJobBatchTimeOut_Reverse.IN := FALSE;

  CASE uiResettingStep OF
            0:
                // Resetting process start

                uiAbortingStep := 0;
                uiAbortedStep  := 0;
				_bRetry := FALSE;

				RoundBeltMoveJob.HandShake.Execute := FALSE;
				RoundBeltMoveJob_Ctrl.Execute := FALSE;
				bAllocateRobotMoveRequest := FALSE;
				DAS_CoreSys.MachineControl.fbAllocateArea.M_ReleaseRoundBeltAccess(E_RoundBeltControlAccess.Allocating);

                IF M_CheckClipsNoError() AND_THEN
                   M_CheckCylindersNoError()
                THEN
                    // no error -> no need to reset
                    bResettingCompleted := TRUE;
                ELSE
                    uiResettingStep := 1000;
                END_IF

            1000:

//                FOR i := 1 TO GVL.NrOfAllocateCylinder DO
//                    IF THIS^.Clips[i].bError THEN
//                        THIS^.Clips[i].M_Reset('Auto Allocating Job Reset');
//                    END_IF

//                    IF THIS^.cylinders[i].bError THEN
//                        THIS^.cylinders[i].M_Reset('Auto Allocating Job Reset');
//                    END_IF
//                END_FOR
				DAS_CoreSys.MachineControl.fbAllocateArea.M_ReleaseRoundBeltAccess(E_RoundBeltControlAccess.Allocating);
                uiResettingStep := 2000;
			
			2000:
//					IF TurnTable.Motor.Error THEN
//					TurnTable.Motor.Reset();
//				END_IF
				
//				IF  AllocateRobot.axX.Error THEN
//					  AllocateRobot.axX.Reset();
//				END_IF
				
//				IF  AllocateRobot.axY.Error THEN
//					  AllocateRobot.axY.Reset();
//				END_IF
				
//				IF RoundBelt.Motor.Error THEN
//					RoundBelt.Motor.Reset();			
//				END_IF
				uiResettingStep := 9000;
				
            9000:
                // Resetting process is finished
                bResettingCompleted := TRUE;
        END_CASE

        IF bResettingCompleted THEN
            eState := STATE_DORMANT;
        END_IF
END_METHOD

END_FUNCTION_BLOCK

// ---- Library/20_MachineUnits/22_AllocateArea/Service/FB_OutRobot_EmptyBoxMove.TcPOU
FUNCTION_BLOCK FB_OutRobot_EmptyBoxMove EXTENDS FB_ObjectBase_V2
VAR_INPUT
//    Execute    :BOOL;   // True : This prog will start.
//    Abort      :BOOL;   // True : This prog will be abort.
//    Reset      :BOOL;   // True : This prog will be reset.
//    ObjectName :STRING; // Set this fb name(About it's action)
	INPUT            			   : REFERENCE TO ST_InputTable;
	Cylinder   					   : REFERENCE TO UNI_CylinderList;
	Motor      					   : REFERENCE TO UNI_MotorList;
	AutoMode_OutRobotMoveMove : st_AutoMode_ClampingBoxesJob;	
	Cylinders					   : REFERENCE TO ARRAY[0..1] OF FB_Cylinder;
	Clips						   : REFERENCE TO ARRAY[0..1] OF FB_Cylinder;
END_VAR

VAR_OUTPUT
//    Busy    :BOOL;        // True : This prog is running.
//    Done    :BOOL;        // True : Command has been executed.
//    Aborted :BOOL;        // True : This prog is aborted.
//    Error   :BOOL;        // True : This prog has an error.
//    ErrorID :UINT;       // Output ErrorID
//    Status  :T_MaxString; // Output this prog status by string(255bytes)
END_VAR

VAR
//    eState :E_MethodStatus_Basic;
//	uiExecutingStep : UDINT; // This var is used to been controll STATE_EXECUTING process.
//	uiResettingStep : UDINT;
//	uiAbortingStep : UDINT;
//	_Executed :BOOL; // Executing process completed.
//	_Error : BOOL; // FB has an error.
//	_ResetCompleted : BOOL; // FB resetting completed.
//	_AbortCompleted : BOOL; // FB aborting completed.
//	_Abort		: BOOL;
	strStatus	: STRING;
	uiResumeStep : UDINT;
	tonTimeOut   :TON;
	tonTimeDelay   :TON;
	tonLeaveDebounce : TON;	// 1850 箱離開感測器去抖
	iWorkingIndex : INT;
	_UniqueErrorCode :STRING;

	PickingPos	: ARRAY[0..1] OF ST_PositionTable;
	PlacingPos  : ARRAY[0..1] OF ST_PositionTable;
	PressCylinderOnI5			   : REFERENCE TO FB_Cylinder;
	bSyncPick	: BOOL;
	bSyncPlace	: BOOL;
	SensorOnConveyor		   : BIT;
	ConveyorMotor				   : REFERENCE TO FB_Motor;
	UseA	: BOOL;
	UseB	: BOOL;
	// Step 切換偵測 (timer 乾淨重置)
	uiExecutingStep_Last : UDINT;
	// Resume / Pause 機制
	bResumeEnabled : BOOL;	// 由 Reset→Execute 觸發,進 EXECUTING step 0 時消費
	bCanPause : BOOL;		// 當前 step 是否允許暫停
	bPauseLast : BOOL;		// 偵測 Pause 釋放邊緣
	// 雙 clip pick / place 旗標 (取代易誤的 iWorkingIndex 共用)
	bPickedA : BOOL;
	bPickedB : BOOL;
	bPlacedA : BOOL;
	bPlacedB : BOOL;
	// Safety: 夾爪是否正夾著箱 (latched, 1700 閉夾成功→TRUE, 2300 開夾成功→FALSE)
	// 有箱時 abort/recovery 禁止張開 clip,避免任意位置掉箱
	bClipHasBox : ARRAY[0..1] OF BOOL;
	// 浮點座標比較容差 (sync 判斷用),避免 LREAL 直接 `=` 被微誤差誤判
	lrEpsPos 	: LREAL := 0.001;
	
	_bRetry		: BOOL;
	bErrorBlinking : BOOL;
	trigErrorReset : R_TRIG;
	tonErrorResetDelay : TON;
END_VAR

A00_BasicUnits();
SUPER^.A10_StateControl();

ACTION A00_BasicUnits:
// Timer 由各 step 自行呼叫並傳 IN/PT,此處不做 freerun call,
// 避免「IN 殘留 TRUE」造成 step 切換後 timer 不歸零。
END_ACTION

METHOD GetModelState
VAR_OUTPUT
    xDone    :BOOL;
    xBusy    :BOOL;
    xError   :BOOL;
    xAborted :BOOL;
    iErrorID :UDINT;
	UniqueErrorCode : STRING;
END_VAR
xDone    := Done;
xBusy    := Busy;
xError   := Error;
xAborted := Aborted;
iErrorID := ErrorID;
UniqueErrorCode := THIS^.UniqueErrorCode;
END_METHOD

METHOD GetName : STRING
GetName := ObjectName;
END_METHOD

METHOD PRIVATE M_CheckCommand : BOOL
VAR_INPUT
END_VAR
IF NOT AutoMode_OutRobotMoveMove.ClampingInfo.UseClibA
AND NOT AutoMode_OutRobotMoveMove.ClampingInfo.UseClibB THEN
	M_CheckCommand := FALSE;
	strStatus := 'FB_OutRobot_EmptyBoxMove , Wrong Command Neither Clamp was used';
	RETURN;
END_IF

M_CheckCommand := TRUE;
END_METHOD

METHOD PRIVATE M_GetResumeEntryStep : UDINT
VAR_INPUT
	uiErrorStep : UDINT;
END_VAR
// Resume 入口對照表: 錯誤點 → 重新進入的安全 checkpoint
// 原則: 跳回該動作的「重新到位」前置 step,確保位置與夾爪狀態先重建
CASE uiErrorStep OF
	1000, 1100, 1300, 1400:
		M_GetResumeEntryStep := 1000;	// 重發 XY 指令 + 重啟 conveyor
	1500, 1700, 1800, 1850:
		M_GetResumeEntryStep := 1000;	// pick 動作錯誤 → 重發 XY 指令從頭來
	2000, 2100:
		M_GetResumeEntryStep := 2000;	// 重新檢查 TT 角度後再移動到 place
	2200, 2300, 2400:
		M_GetResumeEntryStep := 2000;	// place 動作錯誤 → 重檢 TT 角度 + 重發 XY 指令
	2600:
		M_GetResumeEntryStep := 2600;	// 直接重檢 TT 偵測
ELSE
	M_GetResumeEntryStep := 0;	// fallback: 重跑全流程
END_CASE
END_METHOD

METHOD PRIVATE M_GetWorkingConditions : BOOL
VAR_INPUT
END_VAR
IF AutoMode_OutRobotMoveMove.ClampingInfo.UseClibA THEN
	PickingPos[0] :=FUN_GetPositionTableData('I',5,0);
	PlacingPos[0]:=FUN_GetPositionTableData('R',1,0);
	UseA :=TRUE;
END_IF

IF AutoMode_OutRobotMoveMove.ClampingInfo.UseClibB THEN
	PickingPos[1] :=FUN_GetPositionTableData('I',5,1);
	PlacingPos[1]:=FUN_GetPositionTableData('R',2,1);
	UseB := TRUE;
END_IF

// Sync 判斷一律用浮點容差 (lrEpsPos),避免 LREAL 直接比較被微誤差誤判
bSyncPlace := UseA AND UseB
	AND ABS(PlacingPos[0].X_Pos - PlacingPos[1].X_Pos) < lrEpsPos
	AND ABS(PlacingPos[0].Y_Pos - PlacingPos[1].Y_Pos) < lrEpsPos;

bSyncPick := UseA AND UseB
	AND ABS(PickingPos[0].X_Pos - PickingPos[1].X_Pos) < lrEpsPos
	AND ABS(PickingPos[0].Y_Pos - PickingPos[1].Y_Pos) < lrEpsPos;

PressCylinderOnI5 REF= Cylinder.List.fbDifferentSizeCV_Press2;


ConveyorMotor REF= Motor.List.TransmitDifferentSideCV;

M_GetWorkingConditions := TRUE;
END_METHOD

METHOD PRIVATE M_IsOutRobotAtPos : BOOL
VAR_INPUT
	TargetPos : ST_PositionTable;
END_VAR
VAR
	lTol : LREAL := 0.1;
END_VAR
//lTol := GVL_HMI.Setup.Mechanical.OutRobotPositionTolerance;

M_IsOutRobotAtPos :=
		NOT arAxisCtrl_gb[AxisNo.OutRobot_X].Admin.Axis.Status.Moving
	AND NOT arAxisCtrl_gb[AxisNo.OutRobot_Y].Admin.Axis.Status.Moving
	AND ABS(arAxisCtrl_gb[AxisNo.OutRobot_X].Admin.Axis.NcToPlc.ActPos - TargetPos.X_Pos) < lTol
	AND ABS(arAxisCtrl_gb[AxisNo.OutRobot_Y].Admin.Axis.NcToPlc.ActPos - TargetPos.Y_Pos) < lTol;
END_METHOD

METHOD PRIVATE M_IsTurnTableAtPlaceAngle : BOOL
VAR
	lActPos : LREAL;
	lTol    : LREAL := 0.1;
END_VAR
// Place 前 TurnTable 必須位於 0/90/180/270/360 (任一 station)
// 取絕對值處理負角度 (e.g., -90 → 90, -180 → 180)
lActPos := ABS(arAxisCtrl_gb[AxisNo.TurnTable].Admin.Axis.NcToPlc.ModuloActPos);

M_IsTurnTableAtPlaceAngle :=
	   FUN_CheckInPos(ActPos:=lActPos, TargetPos:=0,   ToleranceRange:=lTol)
	OR FUN_CheckInPos(ActPos:=lActPos, TargetPos:=90,  ToleranceRange:=lTol)
	OR FUN_CheckInPos(ActPos:=lActPos, TargetPos:=180, ToleranceRange:=lTol)
	OR FUN_CheckInPos(ActPos:=lActPos, TargetPos:=270, ToleranceRange:=lTol)
	OR FUN_CheckInPos(ActPos:=lActPos, TargetPos:=360, ToleranceRange:=lTol);
END_METHOD

METHOD PRIVATE M_RecoveryAllObjects : BOOL
VAR_INPUT
END_VAR
VAR 
	i : INT;
END_VAR
FOR i:=0 TO 1 DO
	// Clip: 有箱時絕對不張開 (safety),只清錯
	IF Clips[i].xError THEN
		Clips[i].M_Reset();
	ELSIF NOT bClipHasBox[i] THEN
		Clips[i].M_Retract();
	END_IF
	// Cylinder: 一律抬起 (空爪或有箱都安全)
	IF Cylinders[i].xError THEN
		Cylinders[i].M_Reset();
	ELSE
		Cylinders[i].M_Retract();
	END_IF
END_FOR


IF arAxisCtrl_gb[AxisNo.OutRobot_X].Admin.Axis.Status.Error THEN

	arAxisCtrl_gb[AxisNo.OutRobot_X].Admin.ClearError:= TRUE;
ELSE
	arAxisCtrl_gb[AxisNo.OutRobot_X].Admin.ClearError:= FALSE;
END_IF

IF arAxisCtrl_gb[AxisNo.OutRobot_Y].Admin.Axis.Status.Error THEN

	arAxisCtrl_gb[AxisNo.OutRobot_Y].Admin.ClearError:= TRUE;
ELSE
	arAxisCtrl_gb[AxisNo.OutRobot_Y].Admin.ClearError:= FALSE;
END_IF
END_METHOD

METHOD  M_STATE_ABORTED
VAR_INPUT
END_VAR
IF NOT _bRetry THEN
	ERROR 			:= TRUE;
	Busy    		:= FALSE;
	Aborted 		:= TRUE;
	Status 			:= strStatus;
	uiAbortingStep  := 0;
	_AbortCompleted := TRUE;
END_IF

IF reset THEN
	ERROR 	:= FALSE;
	Aborted := FALSE;
	_bRetry	:= TRUE;
END_IF

IF NOT Execute THEN
	eSTATE:=STATE_RESETTING;
// 續做: Reset+Execute 時設旗標,EXECUTING step 0 會跳到 ResumeStep
ELSIF Execute AND _bRetry AND uiResumeStep > 0 THEN
	Status 	:= '';
	bResumeEnabled := TRUE;
	uiExecutingStep := 0;
	eSTATE:=STATE_EXECUTING;
ELSIF Execute AND _bRetry AND uiResumeStep = 0 THEN
	strStatus := 'FB_OutRobot_EmptyBoxMove, this Error can not retry';
	eSTATE := STATE_ERROR;
END_IF
END_METHOD

METHOD  M_STATE_ABORTING
VAR_INPUT
END_VAR
VAR	 
 i : INT;
	bCylinderCheck: BOOL;
END_VAR
Error := TRUE;

// Timer 歸零
tonTimeOut(IN:=FALSE);
tonTimeDelay(IN:=FALSE);
tonLeaveDebounce(IN:=FALSE);

CASE uiAbortingStep OF
	0 :
		_Abort  := FALSE;
		_bRetry := FALSE;
		bCylinderCheck :=TRUE;
		IF __ISVALIDREF(ConveyorMotor) THEN
			ConveyorMotor.M_MotorStop();
		END_IF

		// Safety: 有箱的 clip 絕對不張開,保留夾持狀態等 resume 或人員處理
		FOR i :=0 TO 1 DO
			IF Clips[i].xError THEN
				Clips[i].M_Reset();
			ELSIF NOT bClipHasBox[i] THEN
				Clips[i].M_Retract();
			END_IF
		END_FOR

		// Cylinder 一律抬起 (空爪或有箱都安全,避免殘留在下位撞機構)
		FOR i :=0 TO 1 DO
			IF Cylinders[i].xError THEN
				Cylinders[i].M_Reset();
			END_IF
			Cylinders[i].M_Retract();
			bCylinderCheck:=bCylinderCheck AND Cylinders[i].InRearPosition;
		END_FOR

		// I5 Press 復位
		IF __ISVALIDREF(PressCylinderOnI5) THEN
			IF PressCylinderOnI5.xError THEN
				PressCylinderOnI5.M_Reset();
			ELSE
				PressCylinderOnI5.M_Retract();
			END_IF
		END_IF

		IF bCylinderCheck THEN
			uiAbortingStep:=9999;
		END_IF
	9999:	_AbortCompleted:=TRUE;
END_CASE

IF NOT Execute THEN
	eState := STATE_RESETTING;
ELSIF Execute AND _AbortCompleted THEN
	eSTATE :=STATE_ABORTED;
END_IF
END_METHOD

METHOD  M_STATE_DONE
VAR_INPUT
END_VAR
Busy 	:= FALSE;
Done	:=TRUE;

IF NOT Execute THEN
	eSTATE:=STATE_RESETTING;
END_IF
END_METHOD

METHOD  M_STATE_DORMANT
VAR_INPUT
END_VAR
Busy            := FALSE;
Done            := FALSE;
Aborted         := FALSE;
Error           := FALSE;
ErrorID         := 0;
Status          := '';
_ResetCompleted := FALSE;
_Error          := FALSE;
_Executed       := FALSE;
_Abort	 :=FALSE;
strStatus := M_FormatManagedStatus(
	AlarmId := GVL_ErrorCode.GC_ALARM_ALC_OUTROBOT_EMPTY,
	InnerMessage := GVL_ErrorCode.GC_MSG_0089);
Status := '';
Error := FALSE;
uiExecutingStep :=uiResettingStep :=0;
// Timer 完整歸零 (用實際 FB call,不是只設屬性)
tonTimeOut(IN:=FALSE);
tonTimeDelay(IN:=FALSE);
tonLeaveDebounce(IN:=FALSE);
uiExecutingStep_Last := 0;
_UniqueErrorCode:='0';
iWorkingIndex :=0;
bSyncPick := FALSE;
bSyncPlace := FALSE;
UseA := FALSE;
UseB :=FALSE;
bPickedA := FALSE;
bPickedB := FALSE;
bPlacedA := FALSE;
bPlacedB := FALSE;
bPauseLast := FALSE;
bCanPause := FALSE;
_bRetry	  := FALSE;
_AbortCompleted := FALSE;
uiAbortingStep  := 0;
bErrorBlinking := FALSE;
tonErrorResetDelay.IN := FALSE;
// 非續做模式才清 ResumeStep 與 ClipHasBox,續做模式保留讓 EXECUTING step 0 判斷
IF NOT bResumeEnabled THEN
	uiResumeStep := 0;
	bClipHasBox[0] := FALSE;
	bClipHasBox[1] := FALSE;
END_IF
// 註: M_RecoveryAllObjects 不放 DORMANT 避免與其他 FB 搶 ClearError,
// 以及避免清掉 bClipHasBox 後誤張爪掉箱。僅 EXECUTING step 0 / RESETTING 呼叫。

IF Execute THEN
	eSTATE:=STATE_EXECUTING;
END_IF
END_METHOD

METHOD  M_STATE_ERROR
VAR_INPUT
END_VAR
ERROR   :=TRUE;
Busy	:=FALSE;
_Error  := FALSE;
Status := strStatus;
IF __ISVALIDREF(ConveyorMotor) THEN
	ConveyorMotor.M_MotorStop();
END_IF

// Reset 上升緣觸發 1 秒 Error 暫滅，之後重新亮回
trigErrorReset(CLK := reset);
IF trigErrorReset.Q THEN
	bErrorBlinking := TRUE;
END_IF

tonErrorResetDelay(IN := bErrorBlinking, PT := T#1S);
IF tonErrorResetDelay.Q THEN
	bErrorBlinking := FALSE;
END_IF

